LIN {X -85.223,Y -27.308,Z -231.114,A -90.000,B 90.000,C 0.000} C_DIS
LIN {X -83.227,Y -27.308,Z -229.864,A -90.000,B 90.000,C 0.000} C_DIS
LIN {X -79.994,Y -27.308,Z -227.837,A -90.000,B 90.000,C 0.000} C_DIS
LIN {X -76.849,Y -27.308,Z -225.880,A -90.000,B 90.000,C 0.000} C_DIS
LIN {X -68.403,Y -27.308,Z -220.902,A -90.000,B 90.000,C 0.000} C_DIS
LIN {X -66.455,Y -27.308,Z -219.796,A -90.000,B 90.000,C 0.000} C_DIS
LIN {X -60.717,Y -27.308,Z -216.545,A -90.000,B 90.000,C 0.000} C_DIS
LIN {X -59.585,Y -27.308,Z -215.913,A -90.000,B 90.000,C 0.000} C_DIS
LIN {X -54.120,Y -27.308,Z -212.892,A -90.000,B 90.000,C 0.000} C_DIS
LIN {X -51.972,Y -27.308,Z -211.724,A -90.000,B 90.000,C 0.000} C_DIS
LIN {X -46.281,Y -27.308,Z -208.611,A -90.000,B 90.000,C 0.000} C_DIS
LIN {X -44.940,Y -27.308,Z -207.894,A -90.000,B 90.000,C 0.000} C_DIS
LIN {X -41.211,Y -27.308,Z -205.831,A -90.000,B 90.000,C 0.000} C_DIS
LIN {X -39.138,Y -27.308,Z -204.699,A -90.000,B 90.000,C 0.000} C_DIS
LIN {X -36.802,Y -27.308,Z -203.366,A -90.000,B 90.000,C 0.000} C_DIS
LIN {X -34.331,Y -27.308,Z -201.960,A -90.000,B 90.000,C 0.000} C_DIS
LIN {X -30.365,Y -27.308,Z -199.567,A -90.000,B 90.000,C 0.000} C_DIS
LIN {X -27.103,Y -27.308,Z -197.441,A -90.000,B 90.000,C 0.000} C_DIS
LIN {X -24.362,Y -27.308,Z -195.502,A -90.000,B 90.000,C 0.000} C_DIS
LIN {X -23.811,Y -27.308,Z -195.108,A -90.000,B 90.000,C 0.000} C_DIS
LIN {X -22.633,Y -27.308,Z -194.200,A -90.000,B 90.000,C 0.000} C_DIS
LIN {X -20.957,Y -27.308,Z -192.878,A -90.000,B 90.000,C 0.000} C_DIS
LIN {X -19.924,Y -27.308,Z -192.013,A -90.000,B 90.000,C 0.000} C_DIS
LIN {X -17.934,Y -27.308,Z -190.290,A -90.000,B 90.000,C 0.000} C_DIS
LIN {X -17.733,Y -27.308,Z -190.109,A -90.000,B 90.000,C 0.000} C_DIS
LIN {X -15.439,Y -27.308,Z -187.960,A -90.000,B 90.000,C 0.000} C_DIS
LIN {X -15.234,Y -27.308,Z -187.762,A -90.000,B 90.000,C 0.000} C_DIS
LIN {X -13.962,Y -27.308,Z -186.449,A -90.000,B 90.000,C 0.000} C_DIS
LIN {X -12.177,Y -27.308,Z -184.664,A -90.000,B 90.000,C 0.000} C_DIS
LIN {X -10.066,Y -27.308,Z -182.306,A -90.000,B 90.000,C 0.000} C_DIS
LIN {X -9.477,Y -27.308,Z -181.655,A -90.000,B 90.000,C 0.000} C_DIS
LIN {X -7.788,Y -27.308,Z -179.586,A -90.000,B 90.000,C 0.000} C_DIS
LIN {X -6.794,Y -27.308,Z -178.283,A -90.000,B 90.000,C 0.000} C_DIS
LIN {X -6.582,Y -27.308,Z -177.987,A -90.000,B 90.000,C 0.000} C_DIS
LIN {X -6.159,Y -27.308,Z -177.338,A -90.000,B 90.000,C 0.000} C_DIS
LIN {X -4.783,Y -27.308,Z -175.273,A -90.000,B 90.000,C 0.000} C_DIS
LIN {X -4.713,Y -27.308,Z -175.159,A -90.000,B 90.000,C 0.000} C_DIS
LIN {X -3.540,Y -27.308,Z -173.039,A -90.000,B 90.000,C 0.000} C_DIS
LIN {X -2.865,Y -27.308,Z -171.671,A -90.000,B 90.000,C 0.000} C_DIS
LIN {X -2.832,Y -27.308,Z -171.590,A -90.000,B 90.000,C 0.000} C_DIS
LIN {X -2.604,Y -27.308,Z -170.921,A -90.000,B 90.000,C 0.000} C_DIS
LIN {X -1.680,Y -27.308,Z -168.354,A -90.000,B 90.000,C 0.000} C_DIS
LIN {X -1.356,Y -27.308,Z -166.665,A -90.000,B 90.000,C 0.000} C_DIS
LIN {X -1.145,Y -27.308,Z -165.329,A -90.000,B 90.000,C 0.000} C_DIS
LIN {X -1.146,Y -27.308,Z -165.323,A -90.000,B 90.000,C 0.000} C_DIS
LIN {X -1.174,Y -27.308,Z -164.878,A -90.000,B 90.000,C 0.000} C_DIS
LIN {X -1.320,Y -27.308,Z -162.962,A -90.000,B 90.000,C 0.000} C_DIS
LIN {X -1.678,Y -27.308,Z -162.121,A -90.000,B 90.000,C 0.000} C_DIS
LIN {X -2.018,Y -27.308,Z -161.227,A -90.000,B 90.000,C 0.000} C_DIS
LIN {X -2.779,Y -27.308,Z -160.228,A -90.000,B 90.000,C 0.000} C_DIS
LIN {X -3.012,Y -27.308,Z -159.916,A -90.000,B 90.000,C 0.000} C_DIS
LIN {X -3.062,Y -27.308,Z -159.845,A -90.000,B 90.000,C 0.000} C_DIS
LIN {X -3.809,Y -27.308,Z -159.198,A -90.000,B 90.000,C 0.000} C_DIS
LIN {X -4.494,Y -27.308,Z -158.553,A -90.000,B 90.000,C 0.000} C_DIS
LIN {X -5.258,Y -27.308,Z -158.041,A -90.000,B 90.000,C 0.000} C_DIS
LIN {X -6.409,Y -27.308,Z -157.185,A -90.000,B 90.000,C 0.000} C_DIS
LIN {X -7.420,Y -27.308,Z -156.518,A -90.000,B 90.000,C 0.000} C_DIS
LIN {X -8.434,Y -27.308,Z -155.815,A -90.000,B 90.000,C 0.000} C_DIS
LIN {X -8.921,Y -27.308,Z -155.486,A -90.000,B 90.000,C 0.000} C_DIS
LIN {X -10.919,Y -27.308,Z -154.124,A -90.000,B 90.000,C 0.000} C_DIS
LIN {X -11.534,Y -27.308,Z -153.660,A -90.000,B 90.000,C 0.000} C_DIS
LIN {X -13.381,Y -27.308,Z -152.360,A -90.000,B 90.000,C 0.000} C_DIS
LIN {X -13.865,Y -27.308,Z -151.978,A -90.000,B 90.000,C 0.000} C_DIS
LIN {X -16.164,Y -27.308,Z -150.260,A -90.000,B 90.000,C 0.000} C_DIS
LIN {X -16.733,Y -27.308,Z -149.790,A -90.000,B 90.000,C 0.000} C_DIS
LIN {X -18.323,Y -27.308,Z -148.512,A -90.000,B 90.000,C 0.000} C_DIS
LIN {X -18.612,Y -27.308,Z -148.282,A -90.000,B 90.000,C 0.000} C_DIS
LIN {X -19.226,Y -27.308,Z -147.818,A -90.000,B 90.000,C 0.000} C_DIS
LIN {X -19.599,Y -27.308,Z -147.522,A -90.000,B 90.000,C 0.000} C_DIS
LIN {X -20.909,Y -27.308,Z -146.394,A -90.000,B 90.000,C 0.000} C_DIS
LIN {X -22.705,Y -27.308,Z -144.892,A -90.000,B 90.000,C 0.000} C_DIS
LIN {X -23.016,Y -27.308,Z -144.647,A -90.000,B 90.000,C 0.000} C_DIS
LIN {X -24.434,Y -27.308,Z -143.351,A -90.000,B 90.000,C 0.000} C_DIS
LIN {X -25.785,Y -27.308,Z -142.145,A -90.000,B 90.000,C 0.000} C_DIS
LIN {X -26.430,Y -27.308,Z -141.592,A -90.000,B 90.000,C 0.000} C_DIS
LIN {X -26.511,Y -27.308,Z -141.523,A -90.000,B 90.000,C 0.000} C_DIS
LIN {X -26.798,Y -27.308,Z -141.263,A -90.000,B 90.000,C 0.000} C_DIS
LIN {X -27.182,Y -27.308,Z -140.891,A -90.000,B 90.000,C 0.000} C_DIS
LIN {X -30.222,Y -27.308,Z -137.840,A -90.000,B 90.000,C 0.000} C_DIS
LIN {X -30.546,Y -27.308,Z -137.455,A -90.000,B 90.000,C 0.000} C_DIS
LIN {X -32.740,Y -27.308,Z -134.749,A -90.000,B 90.000,C 0.000} C_DIS
LIN {X -33.314,Y -27.308,Z -134.051,A -90.000,B 90.000,C 0.000} C_DIS
LIN {X -33.612,Y -27.308,Z -133.614,A -90.000,B 90.000,C 0.000} C_DIS
LIN {X -35.907,Y -27.308,Z -130.179,A -90.000,B 90.000,C 0.000} C_DIS
LIN {X -37.258,Y -27.308,Z -127.712,A -90.000,B 90.000,C 0.000} C_DIS
LIN {X -37.397,Y -27.308,Z -127.454,A -90.000,B 90.000,C 0.000} C_DIS
LIN {X -38.165,Y -27.308,Z -126.016,A -90.000,B 90.000,C 0.000} C_DIS
LIN {X -38.975,Y -27.308,Z -124.190,A -90.000,B 90.000,C 0.000} C_DIS
LIN {X -39.648,Y -27.308,Z -122.652,A -90.000,B 90.000,C 0.000} C_DIS
LIN {X -39.793,Y -27.308,Z -122.312,A -90.000,B 90.000,C 0.000} C_DIS
LIN {X -40.196,Y -27.308,Z -121.317,A -90.000,B 90.000,C 0.000} C_DIS
LIN {X -40.311,Y -27.308,Z -120.980,A -90.000,B 90.000,C 0.000} C_DIS
LIN {X -40.482,Y -27.308,Z -120.456,A -90.000,B 90.000,C 0.000} C_DIS
LIN {X -40.902,Y -27.308,Z -119.024,A -90.000,B 90.000,C 0.000} C_DIS
LIN {X -41.166,Y -27.308,Z -118.090,A -90.000,B 90.000,C 0.000} C_DIS
LIN {X -41.278,Y -27.308,Z -117.687,A -90.000,B 90.000,C 0.000} C_DIS
LIN {X -41.299,Y -27.308,Z -117.605,A -90.000,B 90.000,C 0.000} C_DIS
LIN {X -41.911,Y -27.308,Z -115.570,A -90.000,B 90.000,C 0.000} C_DIS
LIN {X -42.357,Y -27.308,Z -114.398,A -90.000,B 90.000,C 0.000} C_DIS
LIN {X -42.549,Y -27.308,Z -113.916,A -90.000,B 90.000,C 0.000} C_DIS
LIN {X -43.092,Y -27.308,Z -112.840,A -90.000,B 90.000,C 0.000} C_DIS
LIN {X -43.558,Y -27.308,Z -111.969,A -90.000,B 90.000,C 0.000} C_DIS
LIN {X -44.072,Y -27.308,Z -111.153,A -90.000,B 90.000,C 0.000} C_DIS
LIN {X -45.121,Y -27.308,Z -109.594,A -90.000,B 90.000,C 0.000} C_DIS
LIN {X -45.338,Y -27.308,Z -109.287,A -90.000,B 90.000,C 0.000} C_DIS
LIN {X -46.992,Y -27.308,Z -107.075,A -90.000,B 90.000,C 0.000} C_DIS
LIN {X -47.098,Y -27.308,Z -106.927,A -90.000,B 90.000,C 0.000} C_DIS
LIN {X -48.585,Y -27.308,Z -104.967,A -90.000,B 90.000,C 0.000} C_DIS
LIN {X -49.203,Y -27.308,Z -104.208,A -90.000,B 90.000,C 0.000} C_DIS
LIN {X -49.940,Y -27.308,Z -103.250,A -90.000,B 90.000,C 0.000} C_DIS
LIN {X -51.313,Y -27.308,Z -101.558,A -90.000,B 90.000,C 0.000} C_DIS
LIN {X -51.724,Y -27.308,Z -101.045,A -90.000,B 90.000,C 0.000} C_DIS
LIN {X -53.185,Y -27.308,Z -99.120,A -90.000,B 90.000,C 0.000} C_DIS
LIN {X -53.957,Y -27.308,Z -98.076,A -90.000,B 90.000,C 0.000} C_DIS
LIN {X -54.226,Y -27.308,Z -97.727,A -90.000,B 90.000,C 0.000} C_DIS
LIN {X -55.529,Y -27.308,Z -95.927,A -90.000,B 90.000,C 0.000} C_DIS
LIN {X -56.485,Y -27.308,Z -94.658,A -90.000,B 90.000,C 0.000} C_DIS
LIN {X -56.867,Y -27.308,Z -94.134,A -90.000,B 90.000,C 0.000} C_DIS
LIN {X -58.660,Y -27.308,Z -91.749,A -90.000,B 90.000,C 0.000} C_DIS
LIN {X -58.816,Y -27.308,Z -91.546,A -90.000,B 90.000,C 0.000} C_DIS
LIN {X -60.216,Y -27.308,Z -89.639,A -90.000,B 90.000,C 0.000} C_DIS
LIN {X -60.437,Y -27.308,Z -89.333,A -90.000,B 90.000,C 0.000} C_DIS
LIN {X -60.531,Y -27.308,Z -89.209,A -90.000,B 90.000,C 0.000} C_DIS
LIN {X -61.646,Y -27.308,Z -87.834,A -90.000,B 90.000,C 0.000} C_DIS
LIN {X -62.365,Y -27.308,Z -86.929,A -90.000,B 90.000,C 0.000} C_DIS
LIN {X -63.967,Y -27.308,Z -85.103,A -90.000,B 90.000,C 0.000} C_DIS
LIN {X -64.183,Y -27.308,Z -84.856,A -90.000,B 90.000,C 0.000} C_DIS
LIN {X -65.298,Y -27.308,Z -83.619,A -90.000,B 90.000,C 0.000} C_DIS
LIN {X -65.834,Y -27.308,Z -82.993,A -90.000,B 90.000,C 0.000} C_DIS
LIN {X -66.748,Y -27.308,Z -81.917,A -90.000,B 90.000,C 0.000} C_DIS
LIN {X -67.132,Y -27.308,Z -81.454,A -90.000,B 90.000,C 0.000} C_DIS
LIN {X -67.558,Y -27.308,Z -80.989,A -90.000,B 90.000,C 0.000} C_DIS
LIN {X -68.611,Y -27.308,Z -79.786,A -90.000,B 90.000,C 0.000} C_DIS
LIN {X -69.303,Y -27.308,Z -78.987,A -90.000,B 90.000,C 0.000} C_DIS
LIN {X -69.822,Y -27.308,Z -78.380,A -90.000,B 90.000,C 0.000} C_DIS
LIN {X -70.935,Y -27.308,Z -77.008,A -90.000,B 90.000,C 0.000} C_DIS
LIN {X -71.960,Y -27.308,Z -75.857,A -90.000,B 90.000,C 0.000} C_DIS
LIN {X -72.414,Y -27.308,Z -75.329,A -90.000,B 90.000,C 0.000} C_DIS
LIN {X -73.458,Y -27.308,Z -74.204,A -90.000,B 90.000,C 0.000} C_DIS
LIN {X -73.957,Y -27.308,Z -73.750,A -90.000,B 90.000,C 0.000} C_DIS
LIN {X -74.254,Y -27.308,Z -73.492,A -90.000,B 90.000,C 0.000} C_DIS
LIN {X -74.565,Y -27.308,Z -73.279,A -90.000,B 90.000,C 0.000} C_DIS
LIN {X -74.767,Y -27.308,Z -73.138,A -90.000,B 90.000,C 0.000} C_DIS
LIN {X -74.798,Y -27.308,Z -73.125,A -90.000,B 90.000,C 0.000} C_DIS
LIN {X -75.017,Y -27.308,Z -73.097,A -90.000,B 90.000,C 0.000} C_DIS
LIN {X -75.670,Y -27.308,Z -73.073,A -90.000,B 90.000,C 0.000} C_DIS
LIN {X -76.020,Y -27.308,Z -73.070,A -90.000,B 90.000,C 0.000} C_DIS
LIN {X -76.334,Y -27.308,Z -73.065,A -90.000,B 90.000,C 0.000} C_DIS
LIN {X -76.599,Y -27.308,Z -73.057,A -90.000,B 90.000,C 0.000} C_DIS
LIN {X -76.851,Y -27.308,Z -73.043,A -90.000,B 90.000,C 0.000} C_DIS
LIN {X -77.230,Y -27.308,Z -73.013,A -90.000,B 90.000,C 0.000} C_DIS
LIN {X -77.574,Y -27.308,Z -72.983,A -90.000,B 90.000,C 0.000} C_DIS
LIN {X -77.718,Y -27.308,Z -72.968,A -90.000,B 90.000,C 0.000} C_DIS
LIN {X -78.228,Y -27.308,Z -72.885,A -90.000,B 90.000,C 0.000} C_DIS
LIN {X -78.608,Y -27.308,Z -72.796,A -90.000,B 90.000,C 0.000} C_DIS
LIN {X -78.915,Y -27.308,Z -72.710,A -90.000,B 90.000,C 0.000} C_DIS
LIN {X -79.319,Y -27.308,Z -72.586,A -90.000,B 90.000,C 0.000} C_DIS
LIN {X -79.675,Y -27.308,Z -72.471,A -90.000,B 90.000,C 0.000} C_DIS
LIN {X -80.019,Y -27.308,Z -72.348,A -90.000,B 90.000,C 0.000} C_DIS
LIN {X -80.375,Y -27.308,Z -72.185,A -90.000,B 90.000,C 0.000} C_DIS
LIN {X -80.697,Y -27.308,Z -72.027,A -90.000,B 90.000,C 0.000} C_DIS
LIN {X -80.992,Y -27.308,Z -71.848,A -90.000,B 90.000,C 0.000} C_DIS
LIN {X -81.324,Y -27.308,Z -71.641,A -90.000,B 90.000,C 0.000} C_DIS
LIN {X -81.637,Y -27.308,Z -71.388,A -90.000,B 90.000,C 0.000} C_DIS
LIN {X -81.835,Y -27.308,Z -71.211,A -90.000,B 90.000,C 0.000} C_DIS
LIN {X -82.059,Y -27.308,Z -71.022,A -90.000,B 90.000,C 0.000} C_DIS
LIN {X -82.156,Y -27.308,Z -70.939,A -90.000,B 90.000,C 0.000} C_DIS
LIN {X -82.435,Y -27.308,Z -70.649,A -90.000,B 90.000,C 0.000} C_DIS
LIN {X -82.682,Y -27.308,Z -70.318,A -90.000,B 90.000,C 0.000} C_DIS
LIN {X -82.800,Y -27.308,Z -70.155,A -90.000,B 90.000,C 0.000} C_DIS
LIN {X -82.856,Y -27.308,Z -70.085,A -90.000,B 90.000,C 0.000} C_DIS
LIN {X -83.029,Y -27.308,Z -69.840,A -90.000,B 90.000,C 0.000} C_DIS
LIN {X -83.229,Y -27.308,Z -69.490,A -90.000,B 90.000,C 0.000} C_DIS
LIN {X -83.356,Y -27.308,Z -69.184,A -90.000,B 90.000,C 0.000} C_DIS
LIN {X -83.500,Y -27.308,Z -68.887,A -90.000,B 90.000,C 0.000} C_DIS
LIN {X -83.522,Y -27.308,Z -68.835,A -90.000,B 90.000,C 0.000} C_DIS
LIN {X -83.644,Y -27.308,Z -68.492,A -90.000,B 90.000,C 0.000} C_DIS
LIN {X -83.662,Y -27.308,Z -68.425,A -90.000,B 90.000,C 0.000} C_DIS
LIN {X -83.731,Y -27.308,Z -68.129,A -90.000,B 90.000,C 0.000} C_DIS
LIN {X -83.778,Y -27.308,Z -67.975,A -90.000,B 90.000,C 0.000} C_DIS
LIN {X -83.872,Y -27.308,Z -67.562,A -90.000,B 90.000,C 0.000} C_DIS
LIN {X -83.897,Y -27.308,Z -67.322,A -90.000,B 90.000,C 0.000} C_DIS
LIN {X -84.004,Y -27.308,Z -66.971,A -90.000,B 90.000,C 0.000} C_DIS
LIN {X -84.037,Y -27.308,Z -66.849,A -90.000,B 90.000,C 0.000} C_DIS
LIN {X -84.152,Y -27.308,Z -66.309,A -90.000,B 90.000,C 0.000} C_DIS
LIN {X -84.180,Y -27.308,Z -66.154,A -90.000,B 90.000,C 0.000} C_DIS
LIN {X -84.260,Y -27.308,Z -65.657,A -90.000,B 90.000,C 0.000} C_DIS
LIN {X -84.279,Y -27.308,Z -65.543,A -90.000,B 90.000,C 0.000} C_DIS
LIN {X -84.322,Y -27.308,Z -65.297,A -90.000,B 90.000,C 0.000} C_DIS
LIN {X -84.357,Y -27.308,Z -65.124,A -90.000,B 90.000,C 0.000} C_DIS
LIN {X -84.404,Y -27.308,Z -64.967,A -90.000,B 90.000,C 0.000} C_DIS
LIN {X -84.600,Y -27.308,Z -64.383,A -90.000,B 90.000,C 0.000} C_DIS
LIN {X -84.702,Y -27.308,Z -64.055,A -90.000,B 90.000,C 0.000} C_DIS
LIN {X -84.904,Y -27.308,Z -63.276,A -90.000,B 90.000,C 0.000} C_DIS
LIN {X -84.929,Y -27.308,Z -63.196,A -90.000,B 90.000,C 0.000} C_DIS
LIN {X -84.968,Y -27.308,Z -63.107,A -90.000,B 90.000,C 0.000} C_DIS
LIN {X -85.046,Y -27.308,Z -62.905,A -90.000,B 90.000,C 0.000} C_DIS
LIN {X -85.068,Y -27.308,Z -62.858,A -90.000,B 90.000,C 0.000} C_DIS
LIN {X -85.176,Y -27.308,Z -62.700,A -90.000,B 90.000,C 0.000} C_DIS
LIN {X -85.293,Y -27.308,Z -62.562,A -90.000,B 90.000,C 0.000} C_DIS
LIN {X -85.630,Y -27.308,Z -62.148,A -90.000,B 90.000,C 0.000} C_DIS
LIN {X -86.250,Y -27.308,Z -61.521,A -90.000,B 90.000,C 0.000} C_DIS
LIN {X -86.385,Y -27.308,Z -61.384,A -90.000,B 90.000,C 0.000} C_DIS
LIN {X -86.893,Y -27.308,Z -60.912,A -90.000,B 90.000,C 0.000} C_DIS
LIN {X -87.654,Y -27.308,Z -60.199,A -90.000,B 90.000,C 0.000} C_DIS
LIN {X -88.400,Y -27.308,Z -59.530,A -90.000,B 90.000,C 0.000} C_DIS
LIN {X -89.022,Y -27.308,Z -58.966,A -90.000,B 90.000,C 0.000} C_DIS
LIN {X -89.404,Y -27.308,Z -58.604,A -90.000,B 90.000,C 0.000} C_DIS
LIN {X -90.679,Y -27.308,Z -57.368,A -90.000,B 90.000,C 0.000} C_DIS
LIN {X -90.874,Y -27.308,Z -57.173,A -90.000,B 90.000,C 0.000} C_DIS
LIN {X -91.295,Y -27.308,Z -56.741,A -90.000,B 90.000,C 0.000} C_DIS
LIN {X -91.759,Y -27.308,Z -56.238,A -90.000,B 90.000,C 0.000} C_DIS
LIN {X -92.620,Y -27.308,Z -55.242,A -90.000,B 90.000,C 0.000} C_DIS
LIN {X -93.104,Y -27.308,Z -54.609,A -90.000,B 90.000,C 0.000} C_DIS
LIN {X -93.380,Y -27.308,Z -54.235,A -90.000,B 90.000,C 0.000} C_DIS
LIN {X -93.514,Y -27.308,Z -54.050,A -90.000,B 90.000,C 0.000} C_DIS
LIN {X -93.898,Y -27.308,Z -53.393,A -90.000,B 90.000,C 0.000} C_DIS
LIN {X -93.958,Y -27.308,Z -53.276,A -90.000,B 90.000,C 0.000} C_DIS
LIN {X -94.142,Y -27.308,Z -52.904,A -90.000,B 90.000,C 0.000} C_DIS
LIN {X -94.334,Y -27.308,Z -52.418,A -90.000,B 90.000,C 0.000} C_DIS
LIN {X -94.397,Y -27.308,Z -52.255,A -90.000,B 90.000,C 0.000} C_DIS
LIN {X -94.572,Y -27.308,Z -51.708,A -90.000,B 90.000,C 0.000} C_DIS
LIN {X -94.624,Y -27.308,Z -51.540,A -90.000,B 90.000,C 0.000} C_DIS
LIN {X -94.663,Y -27.308,Z -51.261,A -90.000,B 90.000,C 0.000} C_DIS
LIN {X -94.690,Y -27.308,Z -50.989,A -90.000,B 90.000,C 0.000} C_DIS
LIN {X -94.708,Y -27.308,Z -50.849,A -90.000,B 90.000,C 0.000} C_DIS
LIN {X -94.705,Y -27.308,Z -50.520,A -90.000,B 90.000,C 0.000} C_DIS
LIN {X -94.685,Y -27.308,Z -50.284,A -90.000,B 90.000,C 0.000} C_DIS
LIN {X -94.633,Y -27.308,Z -49.971,A -90.000,B 90.000,C 0.000} C_DIS
LIN {X -94.628,Y -27.308,Z -49.914,A -90.000,B 90.000,C 0.000} C_DIS
LIN {X -94.559,Y -27.308,Z -49.687,A -90.000,B 90.000,C 0.000} C_DIS
LIN {X -94.426,Y -27.308,Z -49.421,A -90.000,B 90.000,C 0.000} C_DIS
LIN {X -94.404,Y -27.308,Z -49.356,A -90.000,B 90.000,C 0.000} C_DIS
LIN {X -94.289,Y -27.308,Z -49.148,A -90.000,B 90.000,C 0.000} C_DIS
LIN {X -94.134,Y -27.308,Z -48.970,A -90.000,B 90.000,C 0.000} C_DIS
LIN {X -94.079,Y -27.308,Z -48.910,A -90.000,B 90.000,C 0.000} C_DIS
LIN {X -94.043,Y -27.308,Z -48.853,A -90.000,B 90.000,C 0.000} C_DIS
LIN {X -93.887,Y -27.308,Z -48.674,A -90.000,B 90.000,C 0.000} C_DIS
LIN {X -93.617,Y -27.308,Z -48.473,A -90.000,B 90.000,C 0.000} C_DIS
LIN {X -93.557,Y -27.308,Z -48.413,A -90.000,B 90.000,C 0.000} C_DIS
LIN {X -93.414,Y -27.308,Z -48.295,A -90.000,B 90.000,C 0.000} C_DIS
LIN {X -93.204,Y -27.308,Z -48.138,A -90.000,B 90.000,C 0.000} C_DIS
LIN {X -92.952,Y -27.308,Z -48.011,A -90.000,B 90.000,C 0.000} C_DIS
LIN {X -92.775,Y -27.308,Z -47.952,A -90.000,B 90.000,C 0.000} C_DIS
LIN {X -92.483,Y -27.308,Z -47.821,A -90.000,B 90.000,C 0.000} C_DIS
LIN {X -92.213,Y -27.308,Z -47.741,A -90.000,B 90.000,C 0.000} C_DIS
LIN {X -91.652,Y -27.308,Z -47.616,A -90.000,B 90.000,C 0.000} C_DIS
LIN {X -91.311,Y -27.308,Z -47.593,A -90.000,B 90.000,C 0.000} C_DIS
LIN {X -90.543,Y -27.308,Z -47.616,A -90.000,B 90.000,C 0.000} C_DIS
LIN {X -90.225,Y -27.308,Z -47.643,A -90.000,B 90.000,C 0.000} C_DIS
LIN {X -89.409,Y -27.308,Z -47.720,A -90.000,B 90.000,C 0.000} C_DIS
LIN {X -88.277,Y -27.308,Z -47.951,A -90.000,B 90.000,C 0.000} C_DIS
LIN {X -88.112,Y -27.308,Z -47.999,A -90.000,B 90.000,C 0.000} C_DIS
LIN {X -86.815,Y -27.308,Z -48.411,A -90.000,B 90.000,C 0.000} C_DIS
LIN {X -86.455,Y -27.308,Z -48.530,A -90.000,B 90.000,C 0.000} C_DIS
LIN {X -85.645,Y -27.308,Z -48.823,A -90.000,B 90.000,C 0.000} C_DIS
LIN {X -85.388,Y -27.308,Z -48.929,A -90.000,B 90.000,C 0.000} C_DIS
LIN {X -84.854,Y -27.308,Z -49.164,A -90.000,B 90.000,C 0.000} C_DIS
LIN {X -82.923,Y -27.308,Z -50.118,A -90.000,B 90.000,C 0.000} C_DIS
LIN {X -82.842,Y -27.308,Z -50.159,A -90.000,B 90.000,C 0.000} C_DIS
LIN {X -81.799,Y -27.308,Z -50.772,A -90.000,B 90.000,C 0.000} C_DIS
LIN {X -80.820,Y -27.308,Z -51.324,A -90.000,B 90.000,C 0.000} C_DIS
LIN {X -80.098,Y -27.308,Z -51.785,A -90.000,B 90.000,C 0.000} C_DIS
LIN {X -79.415,Y -27.308,Z -52.233,A -90.000,B 90.000,C 0.000} C_DIS
LIN {X -78.943,Y -27.308,Z -52.512,A -90.000,B 90.000,C 0.000} C_DIS
LIN {X -78.820,Y -27.308,Z -52.591,A -90.000,B 90.000,C 0.000} C_DIS
LIN {X -78.713,Y -27.308,Z -52.652,A -90.000,B 90.000,C 0.000} C_DIS
LIN {X -78.353,Y -27.308,Z -52.874,A -90.000,B 90.000,C 0.000} C_DIS
LIN {X -78.152,Y -27.308,Z -52.915,A -90.000,B 90.000,C 0.000} C_DIS
LIN {X -77.685,Y -27.308,Z -52.891,A -90.000,B 90.000,C 0.000} C_DIS
LIN {X -77.521,Y -27.308,Z -52.843,A -90.000,B 90.000,C 0.000} C_DIS
LIN {X -76.977,Y -27.308,Z -52.661,A -90.000,B 90.000,C 0.000} C_DIS
LIN {X -76.822,Y -27.308,Z -52.584,A -90.000,B 90.000,C 0.000} C_DIS
LIN {X -76.230,Y -27.308,Z -52.231,A -90.000,B 90.000,C 0.000} C_DIS
LIN {X -75.911,Y -27.308,Z -51.880,A -90.000,B 90.000,C 0.000} C_DIS
LIN {X -75.721,Y -27.308,Z -51.738,A -90.000,B 90.000,C 0.000} C_DIS
LIN {X -75.688,Y -27.308,Z -51.716,A -90.000,B 90.000,C 0.000} C_DIS
LIN {X -75.432,Y -27.308,Z -51.196,A -90.000,B 90.000,C 0.000} C_DIS
LIN {X -75.358,Y -27.308,Z -51.059,A -90.000,B 90.000,C 0.000} C_DIS
LIN {X -75.315,Y -27.308,Z -51.015,A -90.000,B 90.000,C 0.000} C_DIS
LIN {X -75.268,Y -27.308,Z -50.824,A -90.000,B 90.000,C 0.000} C_DIS
LIN {X -75.257,Y -27.308,Z -50.431,A -90.000,B 90.000,C 0.000} C_DIS
LIN {X -75.437,Y -27.308,Z -49.585,A -90.000,B 90.000,C 0.000} C_DIS
LIN {X -75.451,Y -27.308,Z -49.419,A -90.000,B 90.000,C 0.000} C_DIS
LIN {X -75.470,Y -27.308,Z -49.322,A -90.000,B 90.000,C 0.000} C_DIS
LIN {X -75.528,Y -27.308,Z -48.845,A -90.000,B 90.000,C 0.000} C_DIS
LIN {X -75.614,Y -27.308,Z -48.700,A -90.000,B 90.000,C 0.000} C_DIS
LIN {X -75.778,Y -27.308,Z -48.315,A -90.000,B 90.000,C 0.000} C_DIS
LIN {X -75.772,Y -27.308,Z -48.226,A -90.000,B 90.000,C 0.000} C_DIS
LIN {X -75.702,Y -27.308,Z -48.112,A -90.000,B 90.000,C 0.000} C_DIS
LIN {X -75.670,Y -27.308,Z -47.358,A -90.000,B 90.000,C 0.000} C_DIS
LIN {X -75.666,Y -27.308,Z -47.285,A -90.000,B 90.000,C 0.000} C_DIS
LIN {X -75.614,Y -27.308,Z -47.213,A -90.000,B 90.000,C 0.000} C_DIS
LIN {X -75.532,Y -27.308,Z -47.179,A -90.000,B 90.000,C 0.000} C_DIS
LIN {X -74.785,Y -27.308,Z -46.921,A -90.000,B 90.000,C 0.000} C_DIS
LIN {X -74.518,Y -27.308,Z -46.858,A -90.000,B 90.000,C 0.000} C_DIS
LIN {X -74.497,Y -27.308,Z -46.853,A -90.000,B 90.000,C 0.000} C_DIS
LIN {X -74.317,Y -27.308,Z -46.860,A -90.000,B 90.000,C 0.000} C_DIS
LIN {X -74.256,Y -27.308,Z -46.876,A -90.000,B 90.000,C 0.000} C_DIS
LIN {X -72.929,Y -27.308,Z -47.028,A -90.000,B 90.000,C 0.000} C_DIS
LIN {X -72.759,Y -27.308,Z -47.084,A -90.000,B 90.000,C 0.000} C_DIS
LIN {X -72.617,Y -27.308,Z -47.137,A -90.000,B 90.000,C 0.000} C_DIS
LIN {X -71.380,Y -27.308,Z -47.421,A -90.000,B 90.000,C 0.000} C_DIS
LIN {X -71.211,Y -27.308,Z -47.477,A -90.000,B 90.000,C 0.000} C_DIS
LIN {X -71.067,Y -27.308,Z -47.534,A -90.000,B 90.000,C 0.000} C_DIS
LIN {X -69.599,Y -27.308,Z -47.870,A -90.000,B 90.000,C 0.000} C_DIS
LIN {X -69.349,Y -27.308,Z -47.873,A -90.000,B 90.000,C 0.000} C_DIS
LIN {X -67.886,Y -27.308,Z -48.166,A -90.000,B 90.000,C 0.000} C_DIS
LIN {X -67.535,Y -27.308,Z -48.228,A -90.000,B 90.000,C 0.000} C_DIS
LIN {X -67.302,Y -27.308,Z -48.275,A -90.000,B 90.000,C 0.000} C_DIS
LIN {X -67.283,Y -27.308,Z -48.281,A -90.000,B 90.000,C 0.000} C_DIS
LIN {X -66.642,Y -27.308,Z -48.353,A -90.000,B 90.000,C 0.000} C_DIS
LIN {X -64.888,Y -27.308,Z -48.721,A -90.000,B 90.000,C 0.000} C_DIS
LIN {X -64.684,Y -27.308,Z -48.736,A -90.000,B 90.000,C 0.000} C_DIS
LIN {X -64.583,Y -27.308,Z -48.752,A -90.000,B 90.000,C 0.000} C_DIS
LIN {X -63.765,Y -27.308,Z -48.882,A -90.000,B 90.000,C 0.000} C_DIS
LIN {X -62.172,Y -27.308,Z -49.234,A -90.000,B 90.000,C 0.000} C_DIS
LIN {X -61.720,Y -27.308,Z -49.293,A -90.000,B 90.000,C 0.000} C_DIS
LIN {X -60.768,Y -27.308,Z -49.482,A -90.000,B 90.000,C 0.000} C_DIS
LIN {X -60.425,Y -27.308,Z -49.558,A -90.000,B 90.000,C 0.000} C_DIS
LIN {X -59.345,Y -27.308,Z -49.806,A -90.000,B 90.000,C 0.000} C_DIS
LIN {X -58.678,Y -27.308,Z -49.920,A -90.000,B 90.000,C 0.000} C_DIS
LIN {X -58.325,Y -27.308,Z -49.999,A -90.000,B 90.000,C 0.000} C_DIS
LIN {X -56.851,Y -27.308,Z -50.342,A -90.000,B 90.000,C 0.000} C_DIS
LIN {X -56.345,Y -27.308,Z -50.459,A -90.000,B 90.000,C 0.000} C_DIS
LIN {X -55.296,Y -27.308,Z -50.666,A -90.000,B 90.000,C 0.000} C_DIS
LIN {X -53.371,Y -27.308,Z -51.124,A -90.000,B 90.000,C 0.000} C_DIS
LIN {X -53.286,Y -27.308,Z -51.142,A -90.000,B 90.000,C 0.000} C_DIS
LIN {X -53.131,Y -27.308,Z -51.179,A -90.000,B 90.000,C 0.000} C_DIS
LIN {X -51.402,Y -27.308,Z -51.571,A -90.000,B 90.000,C 0.000} C_DIS
LIN {X -50.457,Y -27.308,Z -51.814,A -90.000,B 90.000,C 0.000} C_DIS
LIN {X -49.578,Y -27.308,Z -52.017,A -90.000,B 90.000,C 0.000} C_DIS
LIN {X -48.351,Y -27.308,Z -52.327,A -90.000,B 90.000,C 0.000} C_DIS
LIN {X -47.858,Y -27.308,Z -52.433,A -90.000,B 90.000,C 0.000} C_DIS
LIN {X -47.456,Y -27.308,Z -52.528,A -90.000,B 90.000,C 0.000} C_DIS
LIN {X -47.282,Y -27.308,Z -52.565,A -90.000,B 90.000,C 0.000} C_DIS
LIN {X -46.851,Y -27.308,Z -52.617,A -90.000,B 90.000,C 0.000} C_DIS
LIN {X -46.055,Y -27.308,Z -52.645,A -90.000,B 90.000,C 0.000} C_DIS
LIN {X -45.267,Y -27.308,Z -52.678,A -90.000,B 90.000,C 0.000} C_DIS
LIN {X -43.988,Y -27.308,Z -52.715,A -90.000,B 90.000,C 0.000} C_DIS
LIN {X -42.867,Y -27.308,Z -52.774,A -90.000,B 90.000,C 0.000} C_DIS
LIN {X -42.549,Y -27.308,Z -52.801,A -90.000,B 90.000,C 0.000} C_DIS
LIN {X -41.808,Y -27.308,Z -52.875,A -90.000,B 90.000,C 0.000} C_DIS
LIN {X -39.572,Y -27.308,Z -53.109,A -90.000,B 90.000,C 0.000} C_DIS
LIN {X -38.701,Y -27.308,Z -53.242,A -90.000,B 90.000,C 0.000} C_DIS
LIN {X -38.096,Y -27.308,Z -53.337,A -90.000,B 90.000,C 0.000} C_DIS
LIN {X -36.582,Y -27.308,Z -53.593,A -90.000,B 90.000,C 0.000} C_DIS
LIN {X -35.657,Y -27.308,Z -53.760,A -90.000,B 90.000,C 0.000} C_DIS
LIN {X -33.190,Y -27.308,Z -54.250,A -90.000,B 90.000,C 0.000} C_DIS
LIN {X -32.731,Y -27.308,Z -54.338,A -90.000,B 90.000,C 0.000} C_DIS
LIN {X -31.973,Y -27.308,Z -54.494,A -90.000,B 90.000,C 0.000} C_DIS
LIN {X -29.563,Y -27.308,Z -55.034,A -90.000,B 90.000,C 0.000} C_DIS
LIN {X -28.572,Y -27.308,Z -55.243,A -90.000,B 90.000,C 0.000} C_DIS
LIN {X -26.759,Y -27.308,Z -55.630,A -90.000,B 90.000,C 0.000} C_DIS
LIN {X -25.274,Y -27.308,Z -55.904,A -90.000,B 90.000,C 0.000} C_DIS
LIN {X -24.524,Y -27.308,Z -56.024,A -90.000,B 90.000,C 0.000} C_DIS
LIN {X -23.511,Y -27.308,Z -56.150,A -90.000,B 90.000,C 0.000} C_DIS
LIN {X -22.723,Y -27.308,Z -56.207,A -90.000,B 90.000,C 0.000} C_DIS
LIN {X -22.397,Y -27.308,Z -56.214,A -90.000,B 90.000,C 0.000} C_DIS
LIN {X -21.650,Y -27.308,Z -56.177,A -90.000,B 90.000,C 0.000} C_DIS
LIN {X -21.553,Y -27.308,Z -56.165,A -90.000,B 90.000,C 0.000} C_DIS
LIN {X -20.887,Y -27.308,Z -56.039,A -90.000,B 90.000,C 0.000} C_DIS
LIN {X -20.751,Y -27.308,Z -56.012,A -90.000,B 90.000,C 0.000} C_DIS
LIN {X -19.986,Y -27.308,Z -55.706,A -90.000,B 90.000,C 0.000} C_DIS
LIN {X -19.512,Y -27.308,Z -55.554,A -90.000,B 90.000,C 0.000} C_DIS
LIN {X -18.660,Y -27.308,Z -55.186,A -90.000,B 90.000,C 0.000} C_DIS
LIN {X -18.036,Y -27.308,Z -54.936,A -90.000,B 90.000,C 0.000} C_DIS
LIN {X -17.892,Y -27.308,Z -54.873,A -90.000,B 90.000,C 0.000} C_DIS
LIN {X -15.925,Y -27.308,Z -54.124,A -90.000,B 90.000,C 0.000} C_DIS
LIN {X -15.504,Y -27.308,Z -53.994,A -90.000,B 90.000,C 0.000} C_DIS
LIN {X -14.478,Y -27.308,Z -53.726,A -90.000,B 90.000,C 0.000} C_DIS
LIN {X -13.147,Y -27.308,Z -53.413,A -90.000,B 90.000,C 0.000} C_DIS
LIN {X -12.872,Y -27.308,Z -53.351,A -90.000,B 90.000,C 0.000} C_DIS
LIN {X -12.439,Y -27.308,Z -53.269,A -90.000,B 90.000,C 0.000} C_DIS
LIN {X -12.071,Y -27.308,Z -53.231,A -90.000,B 90.000,C 0.000} C_DIS
LIN {X -11.636,Y -27.308,Z -53.190,A -90.000,B 90.000,C 0.000} C_DIS
LIN {X -11.196,Y -27.308,Z -53.158,A -90.000,B 90.000,C 0.000} C_DIS
LIN {X -10.086,Y -27.308,Z -53.119,A -90.000,B 90.000,C 0.000} C_DIS
LIN {X -9.111,Y -27.308,Z -53.076,A -90.000,B 90.000,C 0.000} C_DIS
LIN {X -8.324,Y -27.308,Z -53.066,A -90.000,B 90.000,C 0.000} C_DIS
LIN {X -8.178,Y -27.308,Z -53.071,A -90.000,B 90.000,C 0.000} C_DIS
LIN {X -7.941,Y -27.308,Z -53.086,A -90.000,B 90.000,C 0.000} C_DIS
LIN {X -5.929,Y -27.308,Z -53.244,A -90.000,B 90.000,C 0.000} C_DIS
LIN {X -5.507,Y -27.308,Z -53.284,A -90.000,B 90.000,C 0.000} C_DIS
LIN {X -2.491,Y -27.308,Z -53.719,A -90.000,B 90.000,C 0.000} C_DIS
LIN {X -0.877,Y -27.308,Z -54.086,A -90.000,B 90.000,C 0.000} C_DIS
LIN {X -0.384,Y -27.308,Z -54.174,A -90.000,B 90.000,C 0.000} C_DIS
LIN {X 0.435,Y -27.308,Z -54.334,A -90.000,B 90.000,C 0.000} C_DIS
LIN {X 1.127,Y -27.308,Z -54.517,A -90.000,B 90.000,C 0.000} C_DIS
LIN {X 2.471,Y -27.308,Z -54.795,A -90.000,B 90.000,C 0.000} C_DIS
LIN {X 2.756,Y -27.308,Z -54.869,A -90.000,B 90.000,C 0.000} C_DIS
LIN {X 4.090,Y -27.308,Z -55.127,A -90.000,B 90.000,C 0.000} C_DIS
LIN {X 4.736,Y -27.308,Z -55.198,A -90.000,B 90.000,C 0.000} C_DIS
LIN {X 5.276,Y -27.308,Z -55.272,A -90.000,B 90.000,C 0.000} C_DIS
LIN {X 5.687,Y -27.308,Z -55.287,A -90.000,B 90.000,C 0.000} C_DIS
LIN {X 6.858,Y -27.308,Z -55.282,A -90.000,B 90.000,C 0.000} C_DIS
LIN {X 7.864,Y -27.308,Z -55.201,A -90.000,B 90.000,C 0.000} C_DIS
LIN {X 8.134,Y -27.308,Z -55.173,A -90.000,B 90.000,C 0.000} C_DIS
LIN {X 9.252,Y -27.308,Z -55.047,A -90.000,B 90.000,C 0.000} C_DIS
LIN {X 9.652,Y -27.308,Z -55.015,A -90.000,B 90.000,C 0.000} C_DIS
LIN {X 9.923,Y -27.308,Z -54.998,A -90.000,B 90.000,C 0.000} C_DIS
LIN {X 11.157,Y -27.308,Z -55.007,A -90.000,B 90.000,C 0.000} C_DIS
LIN {X 11.508,Y -27.308,Z -55.034,A -90.000,B 90.000,C 0.000} C_DIS
LIN {X 12.331,Y -27.308,Z -55.162,A -90.000,B 90.000,C 0.000} C_DIS
LIN {X 12.569,Y -27.308,Z -55.172,A -90.000,B 90.000,C 0.000} C_DIS
LIN {X 12.876,Y -27.308,Z -55.188,A -90.000,B 90.000,C 0.000} C_DIS
LIN {X 13.561,Y -27.308,Z -55.299,A -90.000,B 90.000,C 0.000} C_DIS
LIN {X 14.134,Y -27.308,Z -55.349,A -90.000,B 90.000,C 0.000} C_DIS
LIN {X 14.781,Y -27.308,Z -55.438,A -90.000,B 90.000,C 0.000} C_DIS
LIN {X 15.213,Y -27.308,Z -55.466,A -90.000,B 90.000,C 0.000} C_DIS
LIN {X 15.445,Y -27.308,Z -55.493,A -90.000,B 90.000,C 0.000} C_DIS
LIN {X 15.887,Y -27.308,Z -55.507,A -90.000,B 90.000,C 0.000} C_DIS
LIN {X 16.274,Y -27.308,Z -55.547,A -90.000,B 90.000,C 0.000} C_DIS
LIN {X 16.722,Y -27.308,Z -55.556,A -90.000,B 90.000,C 0.000} C_DIS
LIN {X 17.040,Y -27.308,Z -55.597,A -90.000,B 90.000,C 0.000} C_DIS
LIN {X 17.121,Y -27.308,Z -55.600,A -90.000,B 90.000,C 0.000} C_DIS
LIN {X 17.542,Y -27.308,Z -55.641,A -90.000,B 90.000,C 0.000} C_DIS
LIN {X 17.858,Y -27.308,Z -55.690,A -90.000,B 90.000,C 0.000} C_DIS
LIN {X 18.015,Y -27.308,Z -55.721,A -90.000,B 90.000,C 0.000} C_DIS
LIN {X 18.204,Y -27.308,Z -55.741,A -90.000,B 90.000,C 0.000} C_DIS
LIN {X 18.617,Y -27.308,Z -55.830,A -90.000,B 90.000,C 0.000} C_DIS
LIN {X 19.037,Y -27.308,Z -55.956,A -90.000,B 90.000,C 0.000} C_DIS
LIN {X 19.207,Y -27.308,Z -55.994,A -90.000,B 90.000,C 0.000} C_DIS
LIN {X 19.430,Y -27.308,Z -55.767,A -90.000,B 90.000,C 0.000} C_DIS
LIN {X 19.513,Y -27.308,Z -55.686,A -90.000,B 90.000,C 0.000} C_DIS
LIN {X 19.879,Y -27.308,Z -55.352,A -90.000,B 90.000,C 0.000} C_DIS
LIN {X 20.370,Y -27.308,Z -54.995,A -90.000,B 90.000,C 0.000} C_DIS
LIN {X 20.445,Y -27.308,Z -54.936,A -90.000,B 90.000,C 0.000} C_DIS
LIN {X 20.628,Y -27.308,Z -54.661,A -90.000,B 90.000,C 0.000} C_DIS
LIN {X 20.626,Y -27.308,Z -54.647,A -90.000,B 90.000,C 0.000} C_DIS
LIN {X 20.641,Y -27.308,Z -54.468,A -90.000,B 90.000,C 0.000} C_DIS
LIN {X 20.652,Y -27.308,Z -54.145,A -90.000,B 90.000,C 0.000} C_DIS
LIN {X 20.672,Y -27.308,Z -53.909,A -90.000,B 90.000,C 0.000} C_DIS
LIN {X 20.840,Y -27.308,Z -53.367,A -90.000,B 90.000,C 0.000} C_DIS
LIN {X 21.056,Y -27.308,Z -52.822,A -90.000,B 90.000,C 0.000} C_DIS
LIN {X 21.165,Y -27.308,Z -52.561,A -90.000,B 90.000,C 0.000} C_DIS
LIN {X 21.317,Y -27.308,Z -52.324,A -90.000,B 90.000,C 0.000} C_DIS
LIN {X 21.558,Y -27.308,Z -51.960,A -90.000,B 90.000,C 0.000} C_DIS
LIN {X 21.711,Y -27.308,Z -51.723,A -90.000,B 90.000,C 0.000} C_DIS
LIN {X 21.853,Y -27.308,Z -51.536,A -90.000,B 90.000,C 0.000} C_DIS
LIN {X 21.956,Y -27.308,Z -51.381,A -90.000,B 90.000,C 0.000} C_DIS
LIN {X 22.023,Y -27.308,Z -51.285,A -90.000,B 90.000,C 0.000} C_DIS
LIN {X 22.445,Y -27.308,Z -50.799,A -90.000,B 90.000,C 0.000} C_DIS
LIN {X 22.741,Y -27.308,Z -50.473,A -90.000,B 90.000,C 0.000} C_DIS
LIN {X 22.835,Y -27.308,Z -50.383,A -90.000,B 90.000,C 0.000} C_DIS
LIN {X 23.027,Y -27.308,Z -50.153,A -90.000,B 90.000,C 0.000} C_DIS
LIN {X 23.258,Y -27.308,Z -49.924,A -90.000,B 90.000,C 0.000} C_DIS
LIN {X 23.576,Y -27.308,Z -49.598,A -90.000,B 90.000,C 0.000} C_DIS
LIN {X 23.818,Y -27.308,Z -49.361,A -90.000,B 90.000,C 0.000} C_DIS
LIN {X 23.864,Y -27.308,Z -49.321,A -90.000,B 90.000,C 0.000} C_DIS
LIN {X 24.021,Y -27.308,Z -49.140,A -90.000,B 90.000,C 0.000} C_DIS
LIN {X 24.598,Y -27.308,Z -48.590,A -90.000,B 90.000,C 0.000} C_DIS
LIN {X 24.869,Y -27.308,Z -48.344,A -90.000,B 90.000,C 0.000} C_DIS
LIN {X 24.954,Y -27.308,Z -48.272,A -90.000,B 90.000,C 0.000} C_DIS
LIN {X 25.011,Y -27.308,Z -48.211,A -90.000,B 90.000,C 0.000} C_DIS
LIN {X 25.672,Y -27.308,Z -47.627,A -90.000,B 90.000,C 0.000} C_DIS
LIN {X 25.884,Y -27.308,Z -47.452,A -90.000,B 90.000,C 0.000} C_DIS
LIN {X 26.341,Y -27.308,Z -47.101,A -90.000,B 90.000,C 0.000} C_DIS
LIN {X 26.504,Y -27.308,Z -46.986,A -90.000,B 90.000,C 0.000} C_DIS
LIN {X 26.644,Y -27.308,Z -46.866,A -90.000,B 90.000,C 0.000} C_DIS
LIN {X 26.996,Y -27.308,Z -46.604,A -90.000,B 90.000,C 0.000} C_DIS
LIN {X 27.661,Y -27.308,Z -46.179,A -90.000,B 90.000,C 0.000} C_DIS
LIN {X 28.096,Y -27.308,Z -45.955,A -90.000,B 90.000,C 0.000} C_DIS
LIN {X 28.319,Y -27.308,Z -45.835,A -90.000,B 90.000,C 0.000} C_DIS
LIN {X 28.417,Y -27.308,Z -45.791,A -90.000,B 90.000,C 0.000} C_DIS
LIN {X 29.159,Y -27.308,Z -45.424,A -90.000,B 90.000,C 0.000} C_DIS
LIN {X 29.587,Y -27.308,Z -45.239,A -90.000,B 90.000,C 0.000} C_DIS
LIN {X 30.107,Y -27.308,Z -45.056,A -90.000,B 90.000,C 0.000} C_DIS
LIN {X 30.247,Y -27.308,Z -45.006,A -90.000,B 90.000,C 0.000} C_DIS
LIN {X 30.342,Y -27.308,Z -44.979,A -90.000,B 90.000,C 0.000} C_DIS
LIN {X 30.800,Y -27.308,Z -44.854,A -90.000,B 90.000,C 0.000} C_DIS
LIN {X 31.703,Y -27.308,Z -44.679,A -90.000,B 90.000,C 0.000} C_DIS
LIN {X 31.904,Y -27.308,Z -44.642,A -90.000,B 90.000,C 0.000} C_DIS
LIN {X 32.382,Y -27.308,Z -44.576,A -90.000,B 90.000,C 0.000} C_DIS
LIN {X 33.026,Y -27.308,Z -44.500,A -90.000,B 90.000,C 0.000} C_DIS
LIN {X 33.299,Y -27.308,Z -44.472,A -90.000,B 90.000,C 0.000} C_DIS
LIN {X 34.106,Y -27.308,Z -44.440,A -90.000,B 90.000,C 0.000} C_DIS
LIN {X 34.379,Y -27.308,Z -44.430,A -90.000,B 90.000,C 0.000} C_DIS
LIN {X 34.809,Y -27.308,Z -44.424,A -90.000,B 90.000,C 0.000} C_DIS
LIN {X 34.908,Y -27.308,Z -44.427,A -90.000,B 90.000,C 0.000} C_DIS
LIN {X 35.661,Y -27.308,Z -44.415,A -90.000,B 90.000,C 0.000} C_DIS
LIN {X 35.944,Y -27.308,Z -44.417,A -90.000,B 90.000,C 0.000} C_DIS
LIN {X 36.401,Y -27.308,Z -44.379,A -90.000,B 90.000,C 0.000} C_DIS
LIN {X 36.864,Y -27.308,Z -44.270,A -90.000,B 90.000,C 0.000} C_DIS
LIN {X 37.986,Y -27.308,Z -43.891,A -90.000,B 90.000,C 0.000} C_DIS
LIN {X 39.146,Y -27.308,Z -43.475,A -90.000,B 90.000,C 0.000} C_DIS
LIN {X 39.665,Y -27.308,Z -43.283,A -90.000,B 90.000,C 0.000} C_DIS
LIN {X 40.086,Y -27.308,Z -43.152,A -90.000,B 90.000,C 0.000} C_DIS
LIN {X 41.064,Y -27.308,Z -42.856,A -90.000,B 90.000,C 0.000} C_DIS
LIN {X 41.887,Y -27.308,Z -42.633,A -90.000,B 90.000,C 0.000} C_DIS
LIN {X 42.587,Y -27.308,Z -42.499,A -90.000,B 90.000,C 0.000} C_DIS
LIN {X 43.328,Y -27.308,Z -42.392,A -90.000,B 90.000,C 0.000} C_DIS
LIN {X 43.780,Y -27.308,Z -42.332,A -90.000,B 90.000,C 0.000} C_DIS
LIN {X 45.231,Y -27.308,Z -42.269,A -90.000,B 90.000,C 0.000} C_DIS
LIN {X 45.687,Y -27.308,Z -42.261,A -90.000,B 90.000,C 0.000} C_DIS
LIN {X 46.114,Y -27.308,Z -42.299,A -90.000,B 90.000,C 0.000} C_DIS
LIN {X 46.490,Y -27.308,Z -42.343,A -90.000,B 90.000,C 0.000} C_DIS
LIN {X 46.845,Y -27.308,Z -42.388,A -90.000,B 90.000,C 0.000} C_DIS
LIN {X 47.882,Y -27.308,Z -42.552,A -90.000,B 90.000,C 0.000} C_DIS
LIN {X 48.337,Y -27.308,Z -42.660,A -90.000,B 90.000,C 0.000} C_DIS
LIN {X 49.744,Y -27.308,Z -43.003,A -90.000,B 90.000,C 0.000} C_DIS
LIN {X 49.923,Y -27.308,Z -43.062,A -90.000,B 90.000,C 0.000} C_DIS
LIN {X 50.341,Y -27.308,Z -43.210,A -90.000,B 90.000,C 0.000} C_DIS
LIN {X 51.412,Y -27.308,Z -43.632,A -90.000,B 90.000,C 0.000} C_DIS
LIN {X 52.285,Y -27.308,Z -44.024,A -90.000,B 90.000,C 0.000} C_DIS
LIN {X 53.027,Y -27.308,Z -44.385,A -90.000,B 90.000,C 0.000} C_DIS
LIN {X 53.452,Y -27.308,Z -44.600,A -90.000,B 90.000,C 0.000} C_DIS
LIN {X 54.382,Y -27.308,Z -45.165,A -90.000,B 90.000,C 0.000} C_DIS
LIN {X 56.073,Y -27.308,Z -46.226,A -90.000,B 90.000,C 0.000} C_DIS
LIN {X 56.461,Y -27.308,Z -46.477,A -90.000,B 90.000,C 0.000} C_DIS
LIN {X 56.666,Y -27.308,Z -46.639,A -90.000,B 90.000,C 0.000} C_DIS
LIN {X 58.184,Y -27.308,Z -47.862,A -90.000,B 90.000,C 0.000} C_DIS
LIN {X 58.556,Y -27.308,Z -48.170,A -90.000,B 90.000,C 0.000} C_DIS
LIN {X 59.100,Y -27.308,Z -48.624,A -90.000,B 90.000,C 0.000} C_DIS
LIN {X 61.179,Y -27.308,Z -50.575,A -90.000,B 90.000,C 0.000} C_DIS
LIN {X 61.864,Y -27.308,Z -51.231,A -90.000,B 90.000,C 0.000} C_DIS
LIN {X 63.171,Y -27.308,Z -52.491,A -90.000,B 90.000,C 0.000} C_DIS
LIN {X 64.048,Y -27.308,Z -53.266,A -90.000,B 90.000,C 0.000} C_DIS
LIN {X 65.006,Y -27.308,Z -54.129,A -90.000,B 90.000,C 0.000} C_DIS
LIN {X 66.147,Y -27.308,Z -54.994,A -90.000,B 90.000,C 0.000} C_DIS
LIN {X 66.886,Y -27.308,Z -55.534,A -90.000,B 90.000,C 0.000} C_DIS
LIN {X 67.739,Y -27.308,Z -56.127,A -90.000,B 90.000,C 0.000} C_DIS
LIN {X 69.016,Y -27.308,Z -56.978,A -90.000,B 90.000,C 0.000} C_DIS
LIN {X 70.300,Y -27.308,Z -57.878,A -90.000,B 90.000,C 0.000} C_DIS
LIN {X 71.059,Y -27.308,Z -58.388,A -90.000,B 90.000,C 0.000} C_DIS
LIN {X 72.700,Y -27.308,Z -59.679,A -90.000,B 90.000,C 0.000} C_DIS
LIN {X 73.132,Y -27.308,Z -60.013,A -90.000,B 90.000,C 0.000} C_DIS
LIN {X 73.257,Y -27.308,Z -60.130,A -90.000,B 90.000,C 0.000} C_DIS
LIN {X 73.889,Y -27.308,Z -60.744,A -90.000,B 90.000,C 0.000} C_DIS
LIN {X 74.937,Y -27.308,Z -61.813,A -90.000,B 90.000,C 0.000} C_DIS
LIN {X 75.234,Y -27.308,Z -62.168,A -90.000,B 90.000,C 0.000} C_DIS
LIN {X 76.071,Y -27.308,Z -63.244,A -90.000,B 90.000,C 0.000} C_DIS
LIN {X 76.407,Y -27.308,Z -63.686,A -90.000,B 90.000,C 0.000} C_DIS
LIN {X 77.071,Y -27.308,Z -64.685,A -90.000,B 90.000,C 0.000} C_DIS
LIN {X 77.643,Y -27.308,Z -65.550,A -90.000,B 90.000,C 0.000} C_DIS
LIN {X 78.032,Y -27.308,Z -66.181,A -90.000,B 90.000,C 0.000} C_DIS
LIN {X 78.362,Y -27.308,Z -66.727,A -90.000,B 90.000,C 0.000} C_DIS
LIN {X 78.433,Y -27.308,Z -66.838,A -90.000,B 90.000,C 0.000} C_DIS
LIN {X 78.586,Y -27.308,Z -66.075,A -90.000,B 90.000,C 0.000} C_DIS
LIN {X 79.091,Y -27.308,Z -64.165,A -90.000,B 90.000,C 0.000} C_DIS
LIN {X 79.194,Y -27.308,Z -63.825,A -90.000,B 90.000,C 0.000} C_DIS
LIN {X 79.834,Y -27.308,Z -61.877,A -90.000,B 90.000,C 0.000} C_DIS
LIN {X 80.548,Y -27.308,Z -59.938,A -90.000,B 90.000,C 0.000} C_DIS
LIN {X 80.691,Y -27.308,Z -59.564,A -90.000,B 90.000,C 0.000} C_DIS
LIN {X 80.736,Y -27.308,Z -59.449,A -90.000,B 90.000,C 0.000} C_DIS
LIN {X 80.883,Y -27.308,Z -59.105,A -90.000,B 90.000,C 0.000} C_DIS
LIN {X 81.411,Y -27.308,Z -57.598,A -90.000,B 90.000,C 0.000} C_DIS
LIN {X 81.507,Y -27.308,Z -57.344,A -90.000,B 90.000,C 0.000} C_DIS
LIN {X 82.417,Y -27.308,Z -55.184,A -90.000,B 90.000,C 0.000} C_DIS
LIN {X 82.593,Y -27.308,Z -54.835,A -90.000,B 90.000,C 0.000} C_DIS
LIN {X 82.991,Y -27.308,Z -54.057,A -90.000,B 90.000,C 0.000} C_DIS
LIN {X 83.553,Y -27.308,Z -52.984,A -90.000,B 90.000,C 0.000} C_DIS
LIN {X 83.615,Y -27.308,Z -52.870,A -90.000,B 90.000,C 0.000} C_DIS
LIN {X 84.800,Y -27.308,Z -50.978,A -90.000,B 90.000,C 0.000} C_DIS
LIN {X 85.033,Y -27.308,Z -50.637,A -90.000,B 90.000,C 0.000} C_DIS
LIN {X 86.349,Y -27.308,Z -48.871,A -90.000,B 90.000,C 0.000} C_DIS
LIN {X 86.730,Y -27.308,Z -48.428,A -90.000,B 90.000,C 0.000} C_DIS
LIN {X 88.126,Y -27.308,Z -46.908,A -90.000,B 90.000,C 0.000} C_DIS
LIN {X 88.529,Y -27.308,Z -46.539,A -90.000,B 90.000,C 0.000} C_DIS
LIN {X 89.798,Y -27.308,Z -45.395,A -90.000,B 90.000,C 0.000} C_DIS
LIN {X 90.067,Y -27.308,Z -45.159,A -90.000,B 90.000,C 0.000} C_DIS
LIN {X 91.727,Y -27.308,Z -43.868,A -90.000,B 90.000,C 0.000} C_DIS
LIN {X 92.155,Y -27.308,Z -43.556,A -90.000,B 90.000,C 0.000} C_DIS
LIN {X 93.797,Y -27.308,Z -42.409,A -90.000,B 90.000,C 0.000} C_DIS
LIN {X 95.424,Y -27.308,Z -41.378,A -90.000,B 90.000,C 0.000} C_DIS
LIN {X 95.864,Y -27.308,Z -41.121,A -90.000,B 90.000,C 0.000} C_DIS
LIN {X 97.376,Y -27.308,Z -40.260,A -90.000,B 90.000,C 0.000} C_DIS
LIN {X 97.527,Y -27.308,Z -40.182,A -90.000,B 90.000,C 0.000} C_DIS
LIN {X 98.805,Y -27.308,Z -39.523,A -90.000,B 90.000,C 0.000} C_DIS
LIN {X 100.317,Y -27.308,Z -38.807,A -90.000,B 90.000,C 0.000} C_DIS
LIN {X 102.237,Y -27.308,Z -37.938,A -90.000,B 90.000,C 0.000} C_DIS
LIN {X 103.453,Y -27.308,Z -37.395,A -90.000,B 90.000,C 0.000} C_DIS
LIN {X 104.516,Y -27.308,Z -36.925,A -90.000,B 90.000,C 0.000} C_DIS
LIN {X 105.407,Y -27.308,Z -36.550,A -90.000,B 90.000,C 0.000} C_DIS
LIN {X 106.871,Y -27.308,Z -35.969,A -90.000,B 90.000,C 0.000} C_DIS
LIN {X 107.396,Y -27.308,Z -35.770,A -90.000,B 90.000,C 0.000} C_DIS
LIN {X 107.855,Y -27.308,Z -35.604,A -90.000,B 90.000,C 0.000} C_DIS
LIN {X 108.317,Y -27.308,Z -35.448,A -90.000,B 90.000,C 0.000} C_DIS
LIN {X 108.770,Y -27.308,Z -35.327,A -90.000,B 90.000,C 0.000} C_DIS
LIN {X 109.221,Y -27.308,Z -35.225,A -90.000,B 90.000,C 0.000} C_DIS
LIN {X 109.732,Y -27.308,Z -35.159,A -90.000,B 90.000,C 0.000} C_DIS
LIN {X 110.108,Y -27.308,Z -35.113,A -90.000,B 90.000,C 0.000} C_DIS
LIN {X 110.615,Y -27.308,Z -35.106,A -90.000,B 90.000,C 0.000} C_DIS
LIN {X 110.949,Y -27.308,Z -35.117,A -90.000,B 90.000,C 0.000} C_DIS
LIN {X 111.443,Y -27.308,Z -35.160,A -90.000,B 90.000,C 0.000} C_DIS
LIN {X 112.087,Y -27.308,Z -35.282,A -90.000,B 90.000,C 0.000} C_DIS
LIN {X 112.431,Y -27.308,Z -35.370,A -90.000,B 90.000,C 0.000} C_DIS
LIN {X 112.915,Y -27.308,Z -35.515,A -90.000,B 90.000,C 0.000} C_DIS
LIN {X 113.055,Y -27.308,Z -35.560,A -90.000,B 90.000,C 0.000} C_DIS
LIN {X 113.505,Y -27.308,Z -35.746,A -90.000,B 90.000,C 0.000} C_DIS
LIN {X 113.979,Y -27.308,Z -35.973,A -90.000,B 90.000,C 0.000} C_DIS
LIN {X 114.416,Y -27.308,Z -36.209,A -90.000,B 90.000,C 0.000} C_DIS
LIN {X 114.565,Y -27.308,Z -36.302,A -90.000,B 90.000,C 0.000} C_DIS
LIN {X 114.950,Y -27.308,Z -36.565,A -90.000,B 90.000,C 0.000} C_DIS
LIN {X 115.050,Y -27.308,Z -36.644,A -90.000,B 90.000,C 0.000} C_DIS
LIN {X 115.445,Y -27.308,Z -36.978,A -90.000,B 90.000,C 0.000} C_DIS
LIN {X 115.513,Y -27.308,Z -37.039,A -90.000,B 90.000,C 0.000} C_DIS
LIN {X 115.852,Y -27.308,Z -37.389,A -90.000,B 90.000,C 0.000} C_DIS
LIN {X 116.079,Y -27.308,Z -37.631,A -90.000,B 90.000,C 0.000} C_DIS
LIN {X 116.439,Y -27.308,Z -38.088,A -90.000,B 90.000,C 0.000} C_DIS
LIN {X 116.700,Y -27.308,Z -38.500,A -90.000,B 90.000,C 0.000} C_DIS
LIN {X 116.926,Y -27.308,Z -38.957,A -90.000,B 90.000,C 0.000} C_DIS
LIN {X 117.065,Y -27.308,Z -39.264,A -90.000,B 90.000,C 0.000} C_DIS
LIN {X 117.133,Y -27.308,Z -39.442,A -90.000,B 90.000,C 0.000} C_DIS
LIN {X 117.260,Y -27.308,Z -39.781,A -90.000,B 90.000,C 0.000} C_DIS
LIN {X 117.389,Y -27.308,Z -40.275,A -90.000,B 90.000,C 0.000} C_DIS
LIN {X 117.462,Y -27.308,Z -40.593,A -90.000,B 90.000,C 0.000} C_DIS
LIN {X 117.540,Y -27.308,Z -41.102,A -90.000,B 90.000,C 0.000} C_DIS
LIN {X 117.595,Y -27.308,Z -41.518,A -90.000,B 90.000,C 0.000} C_DIS
LIN {X 117.630,Y -27.308,Z -41.874,A -90.000,B 90.000,C 0.000} C_DIS
LIN {X 117.658,Y -27.308,Z -42.443,A -90.000,B 90.000,C 0.000} C_DIS
LIN {X 117.668,Y -27.308,Z -42.694,A -90.000,B 90.000,C 0.000} C_DIS
LIN {X 117.662,Y -27.308,Z -42.930,A -90.000,B 90.000,C 0.000} C_DIS
LIN {X 117.651,Y -27.308,Z -43.202,A -90.000,B 90.000,C 0.000} C_DIS
LIN {X 117.608,Y -27.308,Z -43.715,A -90.000,B 90.000,C 0.000} C_DIS
LIN {X 117.567,Y -27.308,Z -44.117,A -90.000,B 90.000,C 0.000} C_DIS
LIN {X 117.484,Y -27.308,Z -44.664,A -90.000,B 90.000,C 0.000} C_DIS
LIN {X 117.391,Y -27.308,Z -45.152,A -90.000,B 90.000,C 0.000} C_DIS
LIN {X 117.260,Y -27.308,Z -45.739,A -90.000,B 90.000,C 0.000} C_DIS
LIN {X 117.108,Y -27.308,Z -46.251,A -90.000,B 90.000,C 0.000} C_DIS
LIN {X 116.900,Y -27.308,Z -46.938,A -90.000,B 90.000,C 0.000} C_DIS
LIN {X 116.548,Y -27.308,Z -47.851,A -90.000,B 90.000,C 0.000} C_DIS
LIN {X 116.372,Y -27.308,Z -48.278,A -90.000,B 90.000,C 0.000} C_DIS
LIN {X 115.873,Y -27.308,Z -49.350,A -90.000,B 90.000,C 0.000} C_DIS
LIN {X 115.132,Y -27.308,Z -50.830,A -90.000,B 90.000,C 0.000} C_DIS
LIN {X 114.586,Y -27.308,Z -51.912,A -90.000,B 90.000,C 0.000} C_DIS
LIN {X 113.941,Y -27.308,Z -53.229,A -90.000,B 90.000,C 0.000} C_DIS
LIN {X 113.276,Y -27.308,Z -54.687,A -90.000,B 90.000,C 0.000} C_DIS
LIN {X 112.799,Y -27.308,Z -55.830,A -90.000,B 90.000,C 0.000} C_DIS
LIN {X 112.213,Y -27.308,Z -57.388,A -90.000,B 90.000,C 0.000} C_DIS
LIN {X 111.674,Y -27.308,Z -59.009,A -90.000,B 90.000,C 0.000} C_DIS
LIN {X 111.236,Y -27.308,Z -60.534,A -90.000,B 90.000,C 0.000} C_DIS
LIN {X 110.710,Y -27.308,Z -62.458,A -90.000,B 90.000,C 0.000} C_DIS
LIN {X 110.135,Y -27.308,Z -64.496,A -90.000,B 90.000,C 0.000} C_DIS
LIN {X 109.994,Y -27.308,Z -64.968,A -90.000,B 90.000,C 0.000} C_DIS
LIN {X 109.345,Y -27.308,Z -67.050,A -90.000,B 90.000,C 0.000} C_DIS
LIN {X 108.519,Y -27.308,Z -69.358,A -90.000,B 90.000,C 0.000} C_DIS
LIN {X 107.562,Y -27.308,Z -71.765,A -90.000,B 90.000,C 0.000} C_DIS
LIN {X 107.403,Y -27.308,Z -72.150,A -90.000,B 90.000,C 0.000} C_DIS
LIN {X 106.414,Y -27.308,Z -74.420,A -90.000,B 90.000,C 0.000} C_DIS
LIN {X 105.411,Y -27.308,Z -76.516,A -90.000,B 90.000,C 0.000} C_DIS
LIN {X 104.209,Y -27.308,Z -78.763,A -90.000,B 90.000,C 0.000} C_DIS
LIN {X 103.956,Y -27.308,Z -79.201,A -90.000,B 90.000,C 0.000} C_DIS
LIN {X 103.058,Y -27.308,Z -80.726,A -90.000,B 90.000,C 0.000} C_DIS
LIN {X 102.174,Y -27.308,Z -82.113,A -90.000,B 90.000,C 0.000} C_DIS
LIN {X 99.671,Y -27.308,Z -85.862,A -90.000,B 90.000,C 0.000} C_DIS
LIN {X 99.672,Y -27.308,Z -86.054,A -90.000,B 90.000,C 0.000} C_DIS
LIN {X 99.706,Y -27.308,Z -86.876,A -90.000,B 90.000,C 0.000} C_DIS
LIN {X 99.730,Y -27.308,Z -87.350,A -90.000,B 90.000,C 0.000} C_DIS
LIN {X 99.760,Y -27.308,Z -89.238,A -90.000,B 90.000,C 0.000} C_DIS
LIN {X 99.804,Y -27.308,Z -90.574,A -90.000,B 90.000,C 0.000} C_DIS
LIN {X 99.802,Y -27.308,Z -90.723,A -90.000,B 90.000,C 0.000} C_DIS
LIN {X 99.766,Y -27.308,Z -92.076,A -90.000,B 90.000,C 0.000} C_DIS
LIN {X 99.744,Y -27.308,Z -92.713,A -90.000,B 90.000,C 0.000} C_DIS
LIN {X 99.703,Y -27.308,Z -93.440,A -90.000,B 90.000,C 0.000} C_DIS
LIN {X 99.624,Y -27.308,Z -94.093,A -90.000,B 90.000,C 0.000} C_DIS
LIN {X 99.441,Y -27.308,Z -95.339,A -90.000,B 90.000,C 0.000} C_DIS
LIN {X 99.378,Y -27.308,Z -95.847,A -90.000,B 90.000,C 0.000} C_DIS
LIN {X 99.108,Y -27.308,Z -97.279,A -90.000,B 90.000,C 0.000} C_DIS
LIN {X 99.074,Y -27.308,Z -97.824,A -90.000,B 90.000,C 0.000} C_DIS
LIN {X 99.067,Y -27.308,Z -97.935,A -90.000,B 90.000,C 0.000} C_DIS
LIN {X 98.999,Y -27.308,Z -98.406,A -90.000,B 90.000,C 0.000} C_DIS
LIN {X 98.847,Y -27.308,Z -99.372,A -90.000,B 90.000,C 0.000} C_DIS
LIN {X 98.832,Y -27.308,Z -99.587,A -90.000,B 90.000,C 0.000} C_DIS
LIN {X 98.643,Y -27.308,Z -101.062,A -90.000,B 90.000,C 0.000} C_DIS
LIN {X 98.635,Y -27.308,Z -101.244,A -90.000,B 90.000,C 0.000} C_DIS
LIN {X 98.514,Y -27.308,Z -102.485,A -90.000,B 90.000,C 0.000} C_DIS
LIN {X 98.487,Y -27.308,Z -102.724,A -90.000,B 90.000,C 0.000} C_DIS
LIN {X 98.410,Y -27.308,Z -104.002,A -90.000,B 90.000,C 0.000} C_DIS
LIN {X 98.416,Y -27.308,Z -104.245,A -90.000,B 90.000,C 0.000} C_DIS
LIN {X 98.436,Y -27.308,Z -104.793,A -90.000,B 90.000,C 0.000} C_DIS
LIN {X 98.553,Y -27.308,Z -105.741,A -90.000,B 90.000,C 0.000} C_DIS
LIN {X 98.742,Y -27.308,Z -106.868,A -90.000,B 90.000,C 0.000} C_DIS
LIN {X 98.927,Y -27.308,Z -108.071,A -90.000,B 90.000,C 0.000} C_DIS
LIN {X 98.995,Y -27.308,Z -108.826,A -90.000,B 90.000,C 0.000} C_DIS
LIN {X 99.065,Y -27.308,Z -109.529,A -90.000,B 90.000,C 0.000} C_DIS
LIN {X 99.124,Y -27.308,Z -110.547,A -90.000,B 90.000,C 0.000} C_DIS
LIN {X 99.170,Y -27.308,Z -111.220,A -90.000,B 90.000,C 0.000} C_DIS
LIN {X 99.195,Y -27.308,Z -111.675,A -90.000,B 90.000,C 0.000} C_DIS
LIN {X 99.250,Y -27.308,Z -112.941,A -90.000,B 90.000,C 0.000} C_DIS
LIN {X 99.285,Y -27.308,Z -113.571,A -90.000,B 90.000,C 0.000} C_DIS
LIN {X 99.356,Y -27.308,Z -115.258,A -90.000,B 90.000,C 0.000} C_DIS
LIN {X 99.402,Y -27.308,Z -116.060,A -90.000,B 90.000,C 0.000} C_DIS
LIN {X 99.483,Y -27.308,Z -117.765,A -90.000,B 90.000,C 0.000} C_DIS
LIN {X 99.501,Y -27.308,Z -118.095,A -90.000,B 90.000,C 0.000} C_DIS
LIN {X 99.596,Y -27.308,Z -120.195,A -90.000,B 90.000,C 0.000} C_DIS
LIN {X 99.668,Y -27.308,Z -122.369,A -90.000,B 90.000,C 0.000} C_DIS
LIN {X 99.672,Y -27.308,Z -122.494,A -90.000,B 90.000,C 0.000} C_DIS
LIN {X 99.705,Y -27.308,Z -124.859,A -90.000,B 90.000,C 0.000} C_DIS
LIN {X 99.674,Y -27.308,Z -127.095,A -90.000,B 90.000,C 0.000} C_DIS
LIN {X 99.669,Y -27.308,Z -127.298,A -90.000,B 90.000,C 0.000} C_DIS
LIN {X 99.576,Y -27.308,Z -129.602,A -90.000,B 90.000,C 0.000} C_DIS
LIN {X 99.430,Y -27.308,Z -132.093,A -90.000,B 90.000,C 0.000} C_DIS
LIN {X 99.401,Y -27.308,Z -132.491,A -90.000,B 90.000,C 0.000} C_DIS
LIN {X 99.240,Y -27.308,Z -134.869,A -90.000,B 90.000,C 0.000} C_DIS
LIN {X 99.055,Y -27.308,Z -137.496,A -90.000,B 90.000,C 0.000} C_DIS
LIN {X 99.014,Y -27.308,Z -138.047,A -90.000,B 90.000,C 0.000} C_DIS
LIN {X 98.786,Y -27.308,Z -140.976,A -90.000,B 90.000,C 0.000} C_DIS
LIN {X 98.742,Y -27.308,Z -141.512,A -90.000,B 90.000,C 0.000} C_DIS
LIN {X 98.453,Y -27.308,Z -144.726,A -90.000,B 90.000,C 0.000} C_DIS
LIN {X 98.409,Y -27.308,Z -145.194,A -90.000,B 90.000,C 0.000} C_DIS
LIN {X 98.000,Y -27.308,Z -149.032,A -90.000,B 90.000,C 0.000} C_DIS
LIN {X 97.974,Y -27.308,Z -149.268,A -90.000,B 90.000,C 0.000} C_DIS
LIN {X 97.503,Y -27.308,Z -152.892,A -90.000,B 90.000,C 0.000} C_DIS
LIN {X 97.368,Y -27.308,Z -153.883,A -90.000,B 90.000,C 0.000} C_DIS
LIN {X 96.787,Y -27.308,Z -157.725,A -90.000,B 90.000,C 0.000} C_DIS
LIN {X 96.371,Y -27.308,Z -160.130,A -90.000,B 90.000,C 0.000} C_DIS
LIN {X 96.129,Y -27.308,Z -161.572,A -90.000,B 90.000,C 0.000} C_DIS
LIN {X 95.887,Y -27.308,Z -162.842,A -90.000,B 90.000,C 0.000} C_DIS
LIN {X 95.656,Y -27.308,Z -164.042,A -90.000,B 90.000,C 0.000} C_DIS
LIN {X 95.157,Y -27.308,Z -166.756,A -90.000,B 90.000,C 0.000} C_DIS
LIN {X 94.964,Y -27.308,Z -167.662,A -90.000,B 90.000,C 0.000} C_DIS
LIN {X 94.382,Y -27.308,Z -170.650,A -90.000,B 90.000,C 0.000} C_DIS
LIN {X 94.253,Y -27.308,Z -171.220,A -90.000,B 90.000,C 0.000} C_DIS
LIN {X 94.233,Y -27.308,Z -171.347,A -90.000,B 90.000,C 0.000} C_DIS
LIN {X 93.664,Y -27.308,Z -174.251,A -90.000,B 90.000,C 0.000} C_DIS
LIN {X 93.593,Y -27.308,Z -174.722,A -90.000,B 90.000,C 0.000} C_DIS
LIN {X 93.562,Y -27.308,Z -174.892,A -90.000,B 90.000,C 0.000} C_DIS
LIN {X 93.252,Y -27.308,Z -176.513,A -90.000,B 90.000,C 0.000} C_DIS
LIN {X 93.035,Y -27.308,Z -178.012,A -90.000,B 90.000,C 0.000} C_DIS
LIN {X 92.825,Y -27.308,Z -179.216,A -90.000,B 90.000,C 0.000} C_DIS
LIN {X 92.607,Y -27.308,Z -180.948,A -90.000,B 90.000,C 0.000} C_DIS
LIN {X 92.501,Y -27.308,Z -181.650,A -90.000,B 90.000,C 0.000} C_DIS
LIN {X 92.309,Y -27.308,Z -183.524,A -90.000,B 90.000,C 0.000} C_DIS
LIN {X 92.225,Y -27.308,Z -184.538,A -90.000,B 90.000,C 0.000} C_DIS
LIN {X 92.131,Y -27.308,Z -185.560,A -90.000,B 90.000,C 0.000} C_DIS
LIN {X 92.118,Y -27.308,Z -185.774,A -90.000,B 90.000,C 0.000} C_DIS
LIN {X 91.991,Y -27.308,Z -187.551,A -90.000,B 90.000,C 0.000} C_DIS
LIN {X 91.960,Y -27.308,Z -188.214,A -90.000,B 90.000,C 0.000} C_DIS
LIN {X 91.909,Y -27.308,Z -189.153,A -90.000,B 90.000,C 0.000} C_DIS
LIN {X 91.865,Y -27.308,Z -190.490,A -90.000,B 90.000,C 0.000} C_DIS
LIN {X 91.861,Y -27.308,Z -190.611,A -90.000,B 90.000,C 0.000} C_DIS
LIN {X 91.827,Y -27.308,Z -191.124,A -90.000,B 90.000,C 0.000} C_DIS
LIN {X 91.723,Y -27.308,Z -193.200,A -90.000,B 90.000,C 0.000} C_DIS
LIN {X 91.695,Y -27.308,Z -193.506,A -90.000,B 90.000,C 0.000} C_DIS
LIN {X 91.405,Y -27.308,Z -196.490,A -90.000,B 90.000,C 0.000} C_DIS
LIN {X 91.359,Y -27.308,Z -196.807,A -90.000,B 90.000,C 0.000} C_DIS
LIN {X 90.822,Y -27.308,Z -199.954,A -90.000,B 90.000,C 0.000} C_DIS
LIN {X 90.790,Y -27.308,Z -200.114,A -90.000,B 90.000,C 0.000} C_DIS
LIN {X 89.886,Y -27.308,Z -204.324,A -90.000,B 90.000,C 0.000} C_DIS
LIN {X 88.760,Y -27.308,Z -209.050,A -90.000,B 90.000,C 0.000} C_DIS
LIN {X 88.010,Y -27.308,Z -212.061,A -90.000,B 90.000,C 0.000} C_DIS
LIN {X 87.487,Y -27.308,Z -214.179,A -90.000,B 90.000,C 0.000} C_DIS
LIN {X 86.889,Y -27.308,Z -216.558,A -90.000,B 90.000,C 0.000} C_DIS
LIN {X 85.924,Y -27.308,Z -220.488,A -90.000,B 90.000,C 0.000} C_DIS
LIN {X 84.901,Y -27.308,Z -224.831,A -90.000,B 90.000,C 0.000} C_DIS
LIN {X 84.678,Y -27.308,Z -225.734,A -90.000,B 90.000,C 0.000} C_DIS
LIN {X 83.482,Y -27.308,Z -230.535,A -90.000,B 90.000,C 0.000} C_DIS
LIN {X 83.339,Y -27.308,Z -231.042,A -90.000,B 90.000,C 0.000} C_DIS
LIN {X 81.710,Y -27.308,Z -236.616,A -90.000,B 90.000,C 0.000} C_DIS
LIN {X 80.664,Y -27.308,Z -239.719,A -90.000,B 90.000,C 0.000} C_DIS
LIN {X 79.774,Y -27.308,Z -242.345,A -90.000,B 90.000,C 0.000} C_DIS
LIN {X 79.674,Y -27.308,Z -242.644,A -90.000,B 90.000,C 0.000} C_DIS
LIN {X 79.313,Y -27.308,Z -243.561,A -90.000,B 90.000,C 0.000} C_DIS
LIN {X 79.313,Y -60.000,Z -243.561,A -90.000,B 90.000,C 0.000} C_DIS
LIN {X 99.737,Y -60.000,Z -85.762,A -90.000,B 90.000,C 0.000} C_DIS
LIN {X 99.737,Y -25.308,Z -85.762,A -90.000,B 90.000,C 0.000} C_DIS
LIN {X 99.743,Y -25.309,Z -85.835,A -90.000,B 90.000,C 0.000} C_DIS
LIN {X 99.776,Y -25.311,Z -86.266,A -90.000,B 90.000,C 0.000} C_DIS
LIN {X 99.848,Y -25.312,Z -87.594,A -90.000,B 90.000,C 0.000} C_DIS
LIN {X 99.950,Y -25.318,Z -88.761,A -90.000,B 90.000,C 0.000} C_DIS
LIN {X 99.975,Y -25.320,Z -89.231,A -90.000,B 90.000,C 0.000} C_DIS
LIN {X 99.996,Y -25.320,Z -89.787,A -90.000,B 90.000,C 0.000} C_DIS
LIN {X 100.011,Y -25.319,Z -90.575,A -90.000,B 90.000,C 0.000} C_DIS
LIN {X 100.027,Y -25.324,Z -91.607,A -90.000,B 90.000,C 0.000} C_DIS
LIN {X 100.040,Y -25.327,Z -92.070,A -90.000,B 90.000,C 0.000} C_DIS
LIN {X 100.040,Y -25.327,Z -92.120,A -90.000,B 90.000,C 0.000} C_DIS
LIN {X 99.989,Y -25.325,Z -92.994,A -90.000,B 90.000,C 0.000} C_DIS
LIN {X 99.970,Y -25.327,Z -93.472,A -90.000,B 90.000,C 0.000} C_DIS
LIN {X 99.951,Y -25.332,Z -93.951,A -90.000,B 90.000,C 0.000} C_DIS
LIN {X 99.929,Y -25.337,Z -94.355,A -90.000,B 90.000,C 0.000} C_DIS
LIN {X 99.903,Y -25.338,Z -94.572,A -90.000,B 90.000,C 0.000} C_DIS
LIN {X 99.811,Y -25.344,Z -95.418,A -90.000,B 90.000,C 0.000} C_DIS
LIN {X 99.790,Y -25.352,Z -95.911,A -90.000,B 90.000,C 0.000} C_DIS
LIN {X 99.734,Y -25.359,Z -96.366,A -90.000,B 90.000,C 0.000} C_DIS
LIN {X 99.681,Y -25.360,Z -96.671,A -90.000,B 90.000,C 0.000} C_DIS
LIN {X 99.640,Y -25.381,Z -97.332,A -90.000,B 90.000,C 0.000} C_DIS
LIN {X 99.631,Y -25.381,Z -97.497,A -90.000,B 90.000,C 0.000} C_DIS
LIN {X 99.602,Y -25.381,Z -97.965,A -90.000,B 90.000,C 0.000} C_DIS
LIN {X 99.588,Y -25.385,Z -98.162,A -90.000,B 90.000,C 0.000} C_DIS
LIN {X 99.522,Y -25.408,Z -99.100,A -90.000,B 90.000,C 0.000} C_DIS
LIN {X 99.492,Y -25.409,Z -99.312,A -90.000,B 90.000,C 0.000} C_DIS
LIN {X 99.482,Y -25.413,Z -99.443,A -90.000,B 90.000,C 0.000} C_DIS
LIN {X 99.471,Y -25.413,Z -99.607,A -90.000,B 90.000,C 0.000} C_DIS
LIN {X 99.397,Y -25.432,Z -100.628,A -90.000,B 90.000,C 0.000} C_DIS
LIN {X 99.351,Y -25.432,Z -100.989,A -90.000,B 90.000,C 0.000} C_DIS
LIN {X 99.345,Y -25.436,Z -101.105,A -90.000,B 90.000,C 0.000} C_DIS
LIN {X 99.338,Y -25.436,Z -101.270,A -90.000,B 90.000,C 0.000} C_DIS
LIN {X 99.290,Y -25.453,Z -102.243,A -90.000,B 90.000,C 0.000} C_DIS
LIN {X 99.268,Y -25.453,Z -102.477,A -90.000,B 90.000,C 0.000} C_DIS
LIN {X 99.261,Y -25.466,Z -102.814,A -90.000,B 90.000,C 0.000} C_DIS
LIN {X 99.256,Y -25.475,Z -103.262,A -90.000,B 90.000,C 0.000} C_DIS
LIN {X 99.232,Y -25.479,Z -103.803,A -90.000,B 90.000,C 0.000} C_DIS
LIN {X 99.238,Y -25.487,Z -103.991,A -90.000,B 90.000,C 0.000} C_DIS
LIN {X 99.275,Y -25.496,Z -104.576,A -90.000,B 90.000,C 0.000} C_DIS
LIN {X 99.293,Y -25.502,Z -104.735,A -90.000,B 90.000,C 0.000} C_DIS
LIN {X 99.345,Y -25.503,Z -105.137,A -90.000,B 90.000,C 0.000} C_DIS
LIN {X 99.398,Y -25.505,Z -105.521,A -90.000,B 90.000,C 0.000} C_DIS
LIN {X 99.418,Y -25.508,Z -105.639,A -90.000,B 90.000,C 0.000} C_DIS
LIN {X 99.538,Y -25.509,Z -106.332,A -90.000,B 90.000,C 0.000} C_DIS
LIN {X 99.584,Y -25.509,Z -106.611,A -90.000,B 90.000,C 0.000} C_DIS
LIN {X 99.804,Y -25.512,Z -108.003,A -90.000,B 90.000,C 0.000} C_DIS
LIN {X 99.889,Y -25.516,Z -108.848,A -90.000,B 90.000,C 0.000} C_DIS
LIN {X 99.954,Y -25.518,Z -109.453,A -90.000,B 90.000,C 0.000} C_DIS
LIN {X 100.042,Y -25.525,Z -110.714,A -90.000,B 90.000,C 0.000} C_DIS
LIN {X 100.076,Y -25.528,Z -111.124,A -90.000,B 90.000,C 0.000} C_DIS
LIN {X 100.094,Y -25.528,Z -111.435,A -90.000,B 90.000,C 0.000} C_DIS
LIN {X 100.138,Y -25.532,Z -112.210,A -90.000,B 90.000,C 0.000} C_DIS
LIN {X 100.185,Y -25.541,Z -112.896,A -90.000,B 90.000,C 0.000} C_DIS
LIN {X 100.222,Y -25.542,Z -113.532,A -90.000,B 90.000,C 0.000} C_DIS
LIN {X 100.255,Y -25.545,Z -114.157,A -90.000,B 90.000,C 0.000} C_DIS
LIN {X 100.312,Y -25.557,Z -115.040,A -90.000,B 90.000,C 0.000} C_DIS
LIN {X 100.367,Y -25.564,Z -115.782,A -90.000,B 90.000,C 0.000} C_DIS
LIN {X 100.452,Y -25.572,Z -117.264,A -90.000,B 90.000,C 0.000} C_DIS
LIN {X 100.491,Y -25.578,Z -117.822,A -90.000,B 90.000,C 0.000} C_DIS
LIN {X 100.566,Y -25.584,Z -119.212,A -90.000,B 90.000,C 0.000} C_DIS
LIN {X 100.606,Y -25.589,Z -119.931,A -90.000,B 90.000,C 0.000} C_DIS
LIN {X 100.626,Y -25.591,Z -120.320,A -90.000,B 90.000,C 0.000} C_DIS
LIN {X 100.715,Y -25.602,Z -122.450,A -90.000,B 90.000,C 0.000} C_DIS
LIN {X 100.735,Y -25.609,Z -123.080,A -90.000,B 90.000,C 0.000} C_DIS
LIN {X 100.772,Y -25.617,Z -124.807,A -90.000,B 90.000,C 0.000} C_DIS
LIN {X 100.759,Y -25.626,Z -126.808,A -90.000,B 90.000,C 0.000} C_DIS
LIN {X 100.760,Y -25.629,Z -127.109,A -90.000,B 90.000,C 0.000} C_DIS
LIN {X 100.756,Y -25.629,Z -127.293,A -90.000,B 90.000,C 0.000} C_DIS
LIN {X 100.677,Y -25.640,Z -129.680,A -90.000,B 90.000,C 0.000} C_DIS
LIN {X 100.547,Y -25.650,Z -132.159,A -90.000,B 90.000,C 0.000} C_DIS
LIN {X 100.370,Y -25.660,Z -134.949,A -90.000,B 90.000,C 0.000} C_DIS
LIN {X 100.170,Y -25.667,Z -137.917,A -90.000,B 90.000,C 0.000} C_DIS
LIN {X 99.898,Y -25.676,Z -141.556,A -90.000,B 90.000,C 0.000} C_DIS
LIN {X 99.829,Y -25.679,Z -142.382,A -90.000,B 90.000,C 0.000} C_DIS
LIN {X 99.595,Y -25.690,Z -145.140,A -90.000,B 90.000,C 0.000} C_DIS
LIN {X 99.435,Y -25.706,Z -146.865,A -90.000,B 90.000,C 0.000} C_DIS
LIN {X 99.189,Y -25.720,Z -149.332,A -90.000,B 90.000,C 0.000} C_DIS
LIN {X 99.130,Y -25.723,Z -149.830,A -90.000,B 90.000,C 0.000} C_DIS
LIN {X 98.944,Y -25.734,Z -151.378,A -90.000,B 90.000,C 0.000} C_DIS
LIN {X 98.766,Y -25.758,Z -152.981,A -90.000,B 90.000,C 0.000} C_DIS
LIN {X 98.623,Y -25.760,Z -154.054,A -90.000,B 90.000,C 0.000} C_DIS
LIN {X 98.502,Y -25.768,Z -154.920,A -90.000,B 90.000,C 0.000} C_DIS
LIN {X 98.285,Y -25.801,Z -156.615,A -90.000,B 90.000,C 0.000} C_DIS
LIN {X 98.098,Y -25.803,Z -157.865,A -90.000,B 90.000,C 0.000} C_DIS
LIN {X 97.780,Y -25.856,Z -160.054,A -90.000,B 90.000,C 0.000} C_DIS
LIN {X 97.720,Y -25.861,Z -160.437,A -90.000,B 90.000,C 0.000} C_DIS
LIN {X 97.635,Y -25.862,Z -160.947,A -90.000,B 90.000,C 0.000} C_DIS
LIN {X 97.506,Y -25.876,Z -161.803,A -90.000,B 90.000,C 0.000} C_DIS
LIN {X 97.198,Y -25.930,Z -163.693,A -90.000,B 90.000,C 0.000} C_DIS
LIN {X 97.133,Y -25.939,Z -164.073,A -90.000,B 90.000,C 0.000} C_DIS
LIN {X 97.050,Y -25.941,Z -164.534,A -90.000,B 90.000,C 0.000} C_DIS
LIN {X 96.639,Y -25.987,Z -166.995,A -90.000,B 90.000,C 0.000} C_DIS
LIN {X 96.584,Y -25.997,Z -167.296,A -90.000,B 90.000,C 0.000} C_DIS
LIN {X 96.553,Y -26.006,Z -167.483,A -90.000,B 90.000,C 0.000} C_DIS
LIN {X 96.482,Y -26.017,Z -167.861,A -90.000,B 90.000,C 0.000} C_DIS
LIN {X 96.013,Y -26.069,Z -170.487,A -90.000,B 90.000,C 0.000} C_DIS
LIN {X 95.939,Y -26.086,Z -170.937,A -90.000,B 90.000,C 0.000} C_DIS
LIN {X 95.903,Y -26.096,Z -171.130,A -90.000,B 90.000,C 0.000} C_DIS
LIN {X 95.826,Y -26.109,Z -171.518,A -90.000,B 90.000,C 0.000} C_DIS
LIN {X 95.818,Y -26.109,Z -171.570,A -90.000,B 90.000,C 0.000} C_DIS
LIN {X 95.377,Y -26.155,Z -174.008,A -90.000,B 90.000,C 0.000} C_DIS
LIN {X 95.288,Y -26.176,Z -174.537,A -90.000,B 90.000,C 0.000} C_DIS
LIN {X 95.270,Y -26.178,Z -174.663,A -90.000,B 90.000,C 0.000} C_DIS
LIN {X 95.224,Y -26.178,Z -174.969,A -90.000,B 90.000,C 0.000} C_DIS
LIN {X 95.195,Y -26.180,Z -175.145,A -90.000,B 90.000,C 0.000} C_DIS
LIN {X 94.945,Y -26.207,Z -176.543,A -90.000,B 90.000,C 0.000} C_DIS
LIN {X 94.904,Y -26.216,Z -176.790,A -90.000,B 90.000,C 0.000} C_DIS
LIN {X 94.728,Y -26.238,Z -178.114,A -90.000,B 90.000,C 0.000} C_DIS
LIN {X 94.708,Y -26.239,Z -178.254,A -90.000,B 90.000,C 0.000} C_DIS
LIN {X 94.534,Y -26.258,Z -179.322,A -90.000,B 90.000,C 0.000} C_DIS
LIN {X 94.512,Y -26.263,Z -179.469,A -90.000,B 90.000,C 0.000} C_DIS
LIN {X 94.405,Y -26.275,Z -180.381,A -90.000,B 90.000,C 0.000} C_DIS
LIN {X 94.310,Y -26.285,Z -181.173,A -90.000,B 90.000,C 0.000} C_DIS
LIN {X 94.245,Y -26.292,Z -181.634,A -90.000,B 90.000,C 0.000} C_DIS
LIN {X 94.214,Y -26.299,Z -181.867,A -90.000,B 90.000,C 0.000} C_DIS
LIN {X 94.108,Y -26.311,Z -182.975,A -90.000,B 90.000,C 0.000} C_DIS
LIN {X 94.040,Y -26.316,Z -183.667,A -90.000,B 90.000,C 0.000} C_DIS
LIN {X 93.963,Y -26.324,Z -184.648,A -90.000,B 90.000,C 0.000} C_DIS
LIN {X 93.876,Y -26.337,Z -185.679,A -90.000,B 90.000,C 0.000} C_DIS
LIN {X 93.864,Y -26.335,Z -185.837,A -90.000,B 90.000,C 0.000} C_DIS
LIN {X 93.731,Y -26.326,Z -187.646,A -90.000,B 90.000,C 0.000} C_DIS
LIN {X 93.696,Y -26.316,Z -188.269,A -90.000,B 90.000,C 0.000} C_DIS
LIN {X 93.640,Y -26.308,Z -189.209,A -90.000,B 90.000,C 0.000} C_DIS
LIN {X 93.614,Y -26.297,Z -189.783,A -90.000,B 90.000,C 0.000} C_DIS
LIN {X 93.578,Y -26.283,Z -190.666,A -90.000,B 90.000,C 0.000} C_DIS
LIN {X 93.539,Y -26.277,Z -191.210,A -90.000,B 90.000,C 0.000} C_DIS
LIN {X 93.413,Y -26.241,Z -193.284,A -90.000,B 90.000,C 0.000} C_DIS
LIN {X 93.388,Y -26.240,Z -193.558,A -90.000,B 90.000,C 0.000} C_DIS
LIN {X 93.081,Y -26.201,Z -196.471,A -90.000,B 90.000,C 0.000} C_DIS
LIN {X 93.053,Y -26.195,Z -196.694,A -90.000,B 90.000,C 0.000} C_DIS
LIN {X 92.990,Y -26.190,Z -197.108,A -90.000,B 90.000,C 0.000} C_DIS
LIN {X 92.498,Y -26.188,Z -199.978,A -90.000,B 90.000,C 0.000} C_DIS
LIN {X 92.464,Y -26.185,Z -200.170,A -90.000,B 90.000,C 0.000} C_DIS
LIN {X 92.428,Y -26.183,Z -200.357,A -90.000,B 90.000,C 0.000} C_DIS
LIN {X 91.596,Y -26.180,Z -204.224,A -90.000,B 90.000,C 0.000} C_DIS
LIN {X 91.500,Y -26.177,Z -204.663,A -90.000,B 90.000,C 0.000} C_DIS
LIN {X 91.338,Y -26.177,Z -205.344,A -90.000,B 90.000,C 0.000} C_DIS
LIN {X 90.346,Y -26.150,Z -209.428,A -90.000,B 90.000,C 0.000} C_DIS
LIN {X 89.732,Y -26.138,Z -211.860,A -90.000,B 90.000,C 0.000} C_DIS
LIN {X 89.184,Y -26.119,Z -214.012,A -90.000,B 90.000,C 0.000} C_DIS
LIN {X 89.098,Y -26.117,Z -214.358,A -90.000,B 90.000,C 0.000} C_DIS
LIN {X 88.436,Y -26.100,Z -216.943,A -90.000,B 90.000,C 0.000} C_DIS
LIN {X 88.002,Y -26.084,Z -218.657,A -90.000,B 90.000,C 0.000} C_DIS
LIN {X 87.455,Y -26.073,Z -220.849,A -90.000,B 90.000,C 0.000} C_DIS
LIN {X 86.848,Y -26.048,Z -223.337,A -90.000,B 90.000,C 0.000} C_DIS
LIN {X 86.425,Y -26.036,Z -225.092,A -90.000,B 90.000,C 0.000} C_DIS
LIN {X 86.312,Y -26.032,Z -225.541,A -90.000,B 90.000,C 0.000} C_DIS
LIN {X 85.727,Y -26.012,Z -227.822,A -90.000,B 90.000,C 0.000} C_DIS
LIN {X 84.945,Y -25.995,Z -230.899,A -90.000,B 90.000,C 0.000} C_DIS
LIN {X 84.878,Y -25.995,Z -231.145,A -90.000,B 90.000,C 0.000} C_DIS
LIN {X 84.799,Y -25.993,Z -231.419,A -90.000,B 90.000,C 0.000} C_DIS
LIN {X 84.196,Y -25.990,Z -233.472,A -90.000,B 90.000,C 0.000} C_DIS
LIN {X 83.203,Y -25.999,Z -236.898,A -90.000,B 90.000,C 0.000} C_DIS
LIN {X 83.159,Y -25.996,Z -237.040,A -90.000,B 90.000,C 0.000} C_DIS
LIN {X 82.577,Y -25.994,Z -238.762,A -90.000,B 90.000,C 0.000} C_DIS
LIN {X 81.186,Y -26.013,Z -242.928,A -90.000,B 90.000,C 0.000} C_DIS
LIN {X 81.126,Y -26.008,Z -243.097,A -90.000,B 90.000,C 0.000} C_DIS
LIN {X 81.095,Y -26.006,Z -243.180,A -90.000,B 90.000,C 0.000} C_DIS
LIN {X 80.945,Y -26.006,Z -243.561,A -90.000,B 90.000,C 0.000} C_DIS
LIN {X 80.945,Y -60.000,Z -243.561,A -90.000,B 90.000,C 0.000} C_DIS
LIN {X -104.795,Y -60.000,Z -243.561,A -90.000,B 90.000,C 0.000} C_DIS
LIN {X -104.795,Y -25.633,Z -243.561,A -90.000,B 90.000,C 0.000} C_DIS
LIN {X -104.580,Y -25.520,Z -243.386,A -90.000,B 90.000,C 0.000} C_DIS
LIN {X -104.091,Y -25.422,Z -243.022,A -90.000,B 90.000,C 0.000} C_DIS
LIN {X -102.165,Y -25.409,Z -241.680,A -90.000,B 90.000,C 0.000} C_DIS
LIN {X -101.815,Y -25.404,Z -241.448,A -90.000,B 90.000,C 0.000} C_DIS
LIN {X -101.290,Y -25.403,Z -241.101,A -90.000,B 90.000,C 0.000} C_DIS
LIN {X -99.060,Y -25.404,Z -239.602,A -90.000,B 90.000,C 0.000} C_DIS
LIN {X -94.267,Y -25.387,Z -236.376,A -90.000,B 90.000,C 0.000} C_DIS
LIN {X -94.091,Y -25.386,Z -236.262,A -90.000,B 90.000,C 0.000} C_DIS
LIN {X -91.828,Y -25.387,Z -234.793,A -90.000,B 90.000,C 0.000} C_DIS
LIN {X -86.127,Y -25.376,Z -231.089,A -90.000,B 90.000,C 0.000} C_DIS
LIN {X -85.503,Y -25.372,Z -230.699,A -90.000,B 90.000,C 0.000} C_DIS
LIN {X -83.295,Y -25.371,Z -229.319,A -90.000,B 90.000,C 0.000} C_DIS
LIN {X -81.347,Y -25.369,Z -228.106,A -90.000,B 90.000,C 0.000} C_DIS
LIN {X -77.837,Y -25.369,Z -225.922,A -90.000,B 90.000,C 0.000} C_DIS
LIN {X -77.273,Y -25.368,Z -225.572,A -90.000,B 90.000,C 0.000} C_DIS
LIN {X -70.404,Y -25.378,Z -221.474,A -90.000,B 90.000,C 0.000} C_DIS
LIN {X -68.665,Y -25.380,Z -220.440,A -90.000,B 90.000,C 0.000} C_DIS
LIN {X -63.103,Y -25.397,Z -217.220,A -90.000,B 90.000,C 0.000} C_DIS
LIN {X -62.499,Y -25.398,Z -216.873,A -90.000,B 90.000,C 0.000} C_DIS
LIN {X -60.438,Y -25.404,Z -215.689,A -90.000,B 90.000,C 0.000} C_DIS
LIN {X -57.046,Y -25.418,Z -213.763,A -90.000,B 90.000,C 0.000} C_DIS
LIN {X -53.948,Y -25.434,Z -212.006,A -90.000,B 90.000,C 0.000} C_DIS
LIN {X -52.541,Y -25.439,Z -211.223,A -90.000,B 90.000,C 0.000} C_DIS
LIN {X -47.807,Y -25.466,Z -208.558,A -90.000,B 90.000,C 0.000} C_DIS
LIN {X -46.982,Y -25.468,Z -208.102,A -90.000,B 90.000,C 0.000} C_DIS
LIN {X -45.416,Y -25.476,Z -207.240,A -90.000,B 90.000,C 0.000} C_DIS
LIN {X -41.620,Y -25.499,Z -205.083,A -90.000,B 90.000,C 0.000} C_DIS
LIN {X -40.275,Y -25.510,Z -204.322,A -90.000,B 90.000,C 0.000} C_DIS
LIN {X -39.802,Y -25.512,Z -204.059,A -90.000,B 90.000,C 0.000} C_DIS
LIN {X -39.563,Y -25.515,Z -203.921,A -90.000,B 90.000,C 0.000} C_DIS
LIN {X -36.358,Y -25.534,Z -202.053,A -90.000,B 90.000,C 0.000} C_DIS
LIN {X -35.118,Y -25.536,Z -201.342,A -90.000,B 90.000,C 0.000} C_DIS
LIN {X -34.804,Y -25.541,Z -201.152,A -90.000,B 90.000,C 0.000} C_DIS
LIN {X -32.840,Y -25.550,Z -199.947,A -90.000,B 90.000,C 0.000} C_DIS
LIN {X -31.076,Y -25.555,Z -198.872,A -90.000,B 90.000,C 0.000} C_DIS
LIN {X -30.793,Y -25.562,Z -198.690,A -90.000,B 90.000,C 0.000} C_DIS
LIN {X -29.270,Y -25.566,Z -197.682,A -90.000,B 90.000,C 0.000} C_DIS
LIN {X -27.758,Y -25.572,Z -196.682,A -90.000,B 90.000,C 0.000} C_DIS
LIN {X -27.657,Y -25.575,Z -196.611,A -90.000,B 90.000,C 0.000} C_DIS
LIN {X -25.053,Y -25.595,Z -194.727,A -90.000,B 90.000,C 0.000} C_DIS
LIN {X -24.514,Y -25.598,Z -194.335,A -90.000,B 90.000,C 0.000} C_DIS
LIN {X -24.400,Y -25.602,Z -194.247,A -90.000,B 90.000,C 0.000} C_DIS
LIN {X -23.307,Y -25.615,Z -193.376,A -90.000,B 90.000,C 0.000} C_DIS
LIN {X -21.742,Y -25.634,Z -192.104,A -90.000,B 90.000,C 0.000} C_DIS
LIN {X -21.662,Y -25.637,Z -192.036,A -90.000,B 90.000,C 0.000} C_DIS
LIN {X -20.660,Y -25.655,Z -191.163,A -90.000,B 90.000,C 0.000} C_DIS
LIN {X -18.993,Y -25.678,Z -189.675,A -90.000,B 90.000,C 0.000} C_DIS
LIN {X -18.712,Y -25.688,Z -189.413,A -90.000,B 90.000,C 0.000} C_DIS
LIN {X -18.530,Y -25.692,Z -189.242,A -90.000,B 90.000,C 0.000} C_DIS
LIN {X -17.066,Y -25.719,Z -187.821,A -90.000,B 90.000,C 0.000} C_DIS
LIN {X -16.310,Y -25.736,Z -187.083,A -90.000,B 90.000,C 0.000} C_DIS
LIN {X -16.128,Y -25.741,Z -186.896,A -90.000,B 90.000,C 0.000} C_DIS
LIN {X -14.867,Y -25.755,Z -185.572,A -90.000,B 90.000,C 0.000} C_DIS
LIN {X -14.538,Y -25.762,Z -185.231,A -90.000,B 90.000,C 0.000} C_DIS
LIN {X -13.972,Y -25.779,Z -184.637,A -90.000,B 90.000,C 0.000} C_DIS
LIN {X -13.500,Y -25.792,Z -184.142,A -90.000,B 90.000,C 0.000} C_DIS
LIN {X -13.141,Y -25.812,Z -183.752,A -90.000,B 90.000,C 0.000} C_DIS
LIN {X -12.289,Y -25.823,Z -182.781,A -90.000,B 90.000,C 0.000} C_DIS
LIN {X -11.792,Y -25.835,Z -182.204,A -90.000,B 90.000,C 0.000} C_DIS
LIN {X -10.942,Y -25.859,Z -181.220,A -90.000,B 90.000,C 0.000} C_DIS
LIN {X -10.545,Y -25.888,Z -180.736,A -90.000,B 90.000,C 0.000} C_DIS
LIN {X -8.942,Y -25.951,Z -178.675,A -90.000,B 90.000,C 0.000} C_DIS
LIN {X -8.563,Y -25.957,Z -178.171,A -90.000,B 90.000,C 0.000} C_DIS
LIN {X -8.437,Y -25.960,Z -178.002,A -90.000,B 90.000,C 0.000} C_DIS
LIN {X -8.018,Y -25.991,Z -177.405,A -90.000,B 90.000,C 0.000} C_DIS
LIN {X -7.852,Y -26.000,Z -177.161,A -90.000,B 90.000,C 0.000} C_DIS
LIN {X -7.485,Y -26.006,Z -176.592,A -90.000,B 90.000,C 0.000} C_DIS
LIN {X -7.038,Y -26.015,Z -175.906,A -90.000,B 90.000,C 0.000} C_DIS
LIN {X -6.291,Y -26.046,Z -174.737,A -90.000,B 90.000,C 0.000} C_DIS
LIN {X -6.115,Y -26.065,Z -174.445,A -90.000,B 90.000,C 0.000} C_DIS
LIN {X -6.067,Y -26.070,Z -174.364,A -90.000,B 90.000,C 0.000} C_DIS
LIN {X -5.639,Y -26.084,Z -173.567,A -90.000,B 90.000,C 0.000} C_DIS
LIN {X -4.970,Y -26.127,Z -172.289,A -90.000,B 90.000,C 0.000} C_DIS
LIN {X -4.541,Y -26.135,Z -171.407,A -90.000,B 90.000,C 0.000} C_DIS
LIN {X -4.367,Y -26.156,Z -171.022,A -90.000,B 90.000,C 0.000} C_DIS
LIN {X -4.335,Y -26.156,Z -170.934,A -90.000,B 90.000,C 0.000} C_DIS
LIN {X -4.152,Y -26.157,Z -170.392,A -90.000,B 90.000,C 0.000} C_DIS
LIN {X -3.340,Y -26.184,Z -168.084,A -90.000,B 90.000,C 0.000} C_DIS
LIN {X -3.289,Y -26.198,Z -167.913,A -90.000,B 90.000,C 0.000} C_DIS
LIN {X -3.006,Y -26.206,Z -166.406,A -90.000,B 90.000,C 0.000} C_DIS
LIN {X -2.814,Y -26.193,Z -165.250,A -90.000,B 90.000,C 0.000} C_DIS
LIN {X -2.814,Y -26.190,Z -165.223,A -90.000,B 90.000,C 0.000} C_DIS
LIN {X -2.826,Y -26.188,Z -165.009,A -90.000,B 90.000,C 0.000} C_DIS
LIN {X -2.901,Y -26.168,Z -163.839,A -90.000,B 90.000,C 0.000} C_DIS
LIN {X -2.930,Y -26.156,Z -163.353,A -90.000,B 90.000,C 0.000} C_DIS
LIN {X -3.052,Y -26.074,Z -162.911,A -90.000,B 90.000,C 0.000} C_DIS
LIN {X -3.122,Y -26.069,Z -162.737,A -90.000,B 90.000,C 0.000} C_DIS
LIN {X -3.172,Y -26.068,Z -162.605,A -90.000,B 90.000,C 0.000} C_DIS
LIN {X -3.396,Y -26.057,Z -161.993,A -90.000,B 90.000,C 0.000} C_DIS
LIN {X -3.568,Y -26.003,Z -161.694,A -90.000,B 90.000,C 0.000} C_DIS
LIN {X -3.766,Y -25.941,Z -161.342,A -90.000,B 90.000,C 0.000} C_DIS
LIN {X -3.783,Y -25.941,Z -161.319,A -90.000,B 90.000,C 0.000} C_DIS
LIN {X -4.136,Y -25.924,Z -160.823,A -90.000,B 90.000,C 0.000} C_DIS
LIN {X -4.259,Y -25.898,Z -160.684,A -90.000,B 90.000,C 0.000} C_DIS
LIN {X -4.673,Y -25.815,Z -160.210,A -90.000,B 90.000,C 0.000} C_DIS
LIN {X -4.777,Y -25.795,Z -160.082,A -90.000,B 90.000,C 0.000} C_DIS
LIN {X -5.308,Y -25.791,Z -159.575,A -90.000,B 90.000,C 0.000} C_DIS
LIN {X -5.645,Y -25.753,Z -159.295,A -90.000,B 90.000,C 0.000} C_DIS
LIN {X -5.922,Y -25.714,Z -159.050,A -90.000,B 90.000,C 0.000} C_DIS
LIN {X -6.025,Y -25.702,Z -158.956,A -90.000,B 90.000,C 0.000} C_DIS
LIN {X -6.594,Y -25.702,Z -158.532,A -90.000,B 90.000,C 0.000} C_DIS
LIN {X -7.082,Y -25.688,Z -158.145,A -90.000,B 90.000,C 0.000} C_DIS
LIN {X -7.593,Y -25.656,Z -157.755,A -90.000,B 90.000,C 0.000} C_DIS
LIN {X -8.030,Y -25.643,Z -157.443,A -90.000,B 90.000,C 0.000} C_DIS
LIN {X -8.769,Y -25.631,Z -156.907,A -90.000,B 90.000,C 0.000} C_DIS
LIN {X -9.531,Y -25.608,Z -156.344,A -90.000,B 90.000,C 0.000} C_DIS
LIN {X -10.166,Y -25.596,Z -155.888,A -90.000,B 90.000,C 0.000} C_DIS
LIN {X -11.467,Y -25.562,Z -154.929,A -90.000,B 90.000,C 0.000} C_DIS
LIN {X -11.606,Y -25.561,Z -154.824,A -90.000,B 90.000,C 0.000} C_DIS
LIN {X -12.055,Y -25.552,Z -154.466,A -90.000,B 90.000,C 0.000} C_DIS
LIN {X -13.873,Y -25.517,Z -153.100,A -90.000,B 90.000,C 0.000} C_DIS
LIN {X -13.939,Y -25.515,Z -153.047,A -90.000,B 90.000,C 0.000} C_DIS
LIN {X -14.378,Y -25.510,Z -152.688,A -90.000,B 90.000,C 0.000} C_DIS
LIN {X -16.492,Y -25.483,Z -151.036,A -90.000,B 90.000,C 0.000} C_DIS
LIN {X -16.631,Y -25.479,Z -150.921,A -90.000,B 90.000,C 0.000} C_DIS
LIN {X -17.066,Y -25.477,Z -150.556,A -90.000,B 90.000,C 0.000} C_DIS
LIN {X -18.950,Y -25.465,Z -149.005,A -90.000,B 90.000,C 0.000} C_DIS
LIN {X -19.532,Y -25.455,Z -148.529,A -90.000,B 90.000,C 0.000} C_DIS
LIN {X -19.891,Y -25.449,Z -148.231,A -90.000,B 90.000,C 0.000} C_DIS
LIN {X -20.050,Y -25.444,Z -148.090,A -90.000,B 90.000,C 0.000} C_DIS
LIN {X -21.355,Y -25.430,Z -146.918,A -90.000,B 90.000,C 0.000} C_DIS
LIN {X -22.195,Y -25.417,Z -146.167,A -90.000,B 90.000,C 0.000} C_DIS
LIN {X -23.129,Y -25.404,Z -145.338,A -90.000,B 90.000,C 0.000} C_DIS
LIN {X -23.372,Y -25.393,Z -145.100,A -90.000,B 90.000,C 0.000} C_DIS
LIN {X -25.945,Y -25.346,Z -142.516,A -90.000,B 90.000,C 0.000} C_DIS
LIN {X -26.675,Y -25.331,Z -141.782,A -90.000,B 90.000,C 0.000} C_DIS
LIN {X -27.120,Y -25.320,Z -141.250,A -90.000,B 90.000,C 0.000} C_DIS
LIN {X -27.590,Y -25.314,Z -140.687,A -90.000,B 90.000,C 0.000} C_DIS
LIN {X -28.721,Y -25.309,Z -139.405,A -90.000,B 90.000,C 0.000} C_DIS
LIN {X -29.254,Y -25.308,Z -138.812,A -90.000,B 90.000,C 0.000} C_DIS
LIN {X -29.371,Y -25.308,Z -138.703,A -90.000,B 90.000,C 0.000} C_DIS
LIN {X -29.419,Y -25.308,Z -138.650,A -90.000,B 90.000,C 0.000} C_DIS
LIN {X -29.421,Y -28.521,Z -138.648,A -90.000,B 90.000,C 0.000} C_DIS
LIN {X -29.422,Y -28.546,Z -138.647,A -90.000,B 90.000,C 0.000} C_DIS
LIN {X -29.431,Y -28.594,Z -138.637,A -90.000,B 90.000,C 0.000} C_DIS
LIN {X -29.442,Y -28.628,Z -138.625,A -90.000,B 90.000,C 0.000} C_DIS
LIN {X -29.464,Y -28.671,Z -138.600,A -90.000,B 90.000,C 0.000} C_DIS
LIN {X -29.546,Y -28.756,Z -138.512,A -90.000,B 90.000,C 0.000} C_DIS
LIN {X -29.617,Y -28.793,Z -138.436,A -90.000,B 90.000,C 0.000} C_DIS
LIN {X -29.728,Y -28.808,Z -138.320,A -90.000,B 90.000,C 0.000} C_DIS
LIN {X -29.770,Y -28.796,Z -138.278,A -90.000,B 90.000,C 0.000} C_DIS
LIN {X -29.805,Y -28.775,Z -138.245,A -90.000,B 90.000,C 0.000} C_DIS
LIN {X -29.830,Y -28.748,Z -138.221,A -90.000,B 90.000,C 0.000} C_DIS
LIN {X -29.850,Y -28.717,Z -138.204,A -90.000,B 90.000,C 0.000} C_DIS
LIN {X -29.864,Y -28.682,Z -138.192,A -90.000,B 90.000,C 0.000} C_DIS
LIN {X -29.874,Y -28.643,Z -138.185,A -90.000,B 90.000,C 0.000} C_DIS
LIN {X -29.880,Y -28.600,Z -138.182,A -90.000,B 90.000,C 0.000} C_DIS
LIN {X -29.883,Y -28.550,Z -138.181,A -90.000,B 90.000,C 0.000} C_DIS
LIN {X -29.886,Y -25.306,Z -138.182,A -90.000,B 90.000,C 0.000} C_DIS
LIN {X -29.898,Y -25.308,Z -138.175,A -90.000,B 90.000,C 0.000} C_DIS
LIN {X -29.907,Y -25.308,Z -138.175,A -90.000,B 90.000,C 0.000} C_DIS
LIN {X -29.926,Y -25.308,Z -138.163,A -90.000,B 90.000,C 0.000} C_DIS
LIN {X -29.987,Y -25.308,Z -138.103,A -90.000,B 90.000,C 0.000} C_DIS
LIN {X -30.165,Y -25.308,Z -137.903,A -90.000,B 90.000,C 0.000} C_DIS
LIN {X -30.320,Y -25.307,Z -137.740,A -90.000,B 90.000,C 0.000} C_DIS
LIN {X -30.505,Y -25.308,Z -137.505,A -90.000,B 90.000,C 0.000} C_DIS
LIN {X -30.527,Y -25.308,Z -137.478,A -90.000,B 90.000,C 0.000} C_DIS
LIN {X -30.801,Y -25.308,Z -137.155,A -90.000,B 90.000,C 0.000} C_DIS
LIN {X -31.254,Y -25.308,Z -136.631,A -90.000,B 90.000,C 0.000} C_DIS
LIN {X -31.437,Y -25.308,Z -136.424,A -90.000,B 90.000,C 0.000} C_DIS
LIN {X -31.726,Y -25.308,Z -136.106,A -90.000,B 90.000,C 0.000} C_DIS
LIN {X -31.926,Y -25.308,Z -135.899,A -90.000,B 90.000,C 0.000} C_DIS
LIN {X -32.055,Y -25.308,Z -135.778,A -90.000,B 90.000,C 0.000} C_DIS
LIN {X -32.098,Y -25.308,Z -135.743,A -90.000,B 90.000,C 0.000} C_DIS
LIN {X -32.141,Y -25.308,Z -135.715,A -90.000,B 90.000,C 0.000} C_DIS
LIN {X -32.165,Y -25.308,Z -135.707,A -90.000,B 90.000,C 0.000} C_DIS
LIN {X -32.187,Y -25.308,Z -135.715,A -90.000,B 90.000,C 0.000} C_DIS
LIN {X -32.199,Y -25.308,Z -135.705,A -90.000,B 90.000,C 0.000} C_DIS
LIN {X -32.264,Y -25.308,Z -135.615,A -90.000,B 90.000,C 0.000} C_DIS
LIN {X -32.758,Y -25.308,Z -134.874,A -90.000,B 90.000,C 0.000} C_DIS
LIN {X -33.539,Y -25.308,Z -133.722,A -90.000,B 90.000,C 0.000} C_DIS
LIN {X -33.583,Y -25.308,Z -133.658,A -90.000,B 90.000,C 0.000} C_DIS
LIN {X -33.873,Y -25.308,Z -133.234,A -90.000,B 90.000,C 0.000} C_DIS
LIN {X -34.353,Y -25.306,Z -132.544,A -90.000,B 90.000,C 0.000} C_DIS
LIN {X -34.546,Y -25.305,Z -132.271,A -90.000,B 90.000,C 0.000} C_DIS
LIN {X -34.852,Y -25.301,Z -131.850,A -90.000,B 90.000,C 0.000} C_DIS
LIN {X -35.064,Y -25.296,Z -131.572,A -90.000,B 90.000,C 0.000} C_DIS
LIN {X -35.199,Y -25.291,Z -131.408,A -90.000,B 90.000,C 0.000} C_DIS
LIN {X -35.244,Y -25.288,Z -131.359,A -90.000,B 90.000,C 0.000} C_DIS
LIN {X -35.298,Y -25.283,Z -131.310,A -90.000,B 90.000,C 0.000} C_DIS
LIN {X -35.312,Y -25.280,Z -131.302,A -90.000,B 90.000,C 0.000} C_DIS
LIN {X -35.328,Y -25.274,Z -131.303,A -90.000,B 90.000,C 0.000} C_DIS
LIN {X -35.332,Y -25.273,Z -131.299,A -90.000,B 90.000,C 0.000} C_DIS
LIN {X -35.400,Y -25.270,Z -131.166,A -90.000,B 90.000,C 0.000} C_DIS
LIN {X -35.495,Y -25.272,Z -130.977,A -90.000,B 90.000,C 0.000} C_DIS
LIN {X -35.899,Y -25.284,Z -130.208,A -90.000,B 90.000,C 0.000} C_DIS
LIN {X -36.063,Y -25.288,Z -129.916,A -90.000,B 90.000,C 0.000} C_DIS
LIN {X -36.463,Y -25.300,Z -129.178,A -90.000,B 90.000,C 0.000} C_DIS
LIN {X -36.704,Y -25.308,Z -128.724,A -90.000,B 90.000,C 0.000} C_DIS
LIN {X -37.294,Y -25.327,Z -127.647,A -90.000,B 90.000,C 0.000} C_DIS
LIN {X -37.314,Y -25.333,Z -127.610,A -90.000,B 90.000,C 0.000} C_DIS
LIN {X -37.546,Y -25.332,Z -127.187,A -90.000,B 90.000,C 0.000} C_DIS
LIN {X -38.004,Y -25.308,Z -126.352,A -90.000,B 90.000,C 0.000} C_DIS
LIN {X -38.234,Y -25.309,Z -125.927,A -90.000,B 90.000,C 0.000} C_DIS
LIN {X -38.970,Y -25.309,Z -124.276,A -90.000,B 90.000,C 0.000} C_DIS
LIN {X -39.697,Y -25.311,Z -122.799,A -90.000,B 90.000,C 0.000} C_DIS
LIN {X -39.732,Y -25.311,Z -122.727,A -90.000,B 90.000,C 0.000} C_DIS
LIN {X -40.349,Y -25.314,Z -121.319,A -90.000,B 90.000,C 0.000} C_DIS
LIN {X -40.676,Y -25.320,Z -120.569,A -90.000,B 90.000,C 0.000} C_DIS
LIN {X -40.863,Y -25.327,Z -120.128,A -90.000,B 90.000,C 0.000} C_DIS
LIN {X -41.120,Y -25.332,Z -119.369,A -90.000,B 90.000,C 0.000} C_DIS
LIN {X -41.565,Y -25.355,Z -118.259,A -90.000,B 90.000,C 0.000} C_DIS
LIN {X -41.684,Y -25.363,Z -117.960,A -90.000,B 90.000,C 0.000} C_DIS
LIN {X -41.912,Y -25.372,Z -117.299,A -90.000,B 90.000,C 0.000} C_DIS
LIN {X -42.392,Y -25.417,Z -116.229,A -90.000,B 90.000,C 0.000} C_DIS
LIN {X -42.444,Y -25.423,Z -116.111,A -90.000,B 90.000,C 0.000} C_DIS
LIN {X -42.538,Y -25.431,Z -115.883,A -90.000,B 90.000,C 0.000} C_DIS
LIN {X -42.593,Y -25.435,Z -115.747,A -90.000,B 90.000,C 0.000} C_DIS
LIN {X -42.672,Y -25.438,Z -115.558,A -90.000,B 90.000,C 0.000} C_DIS
LIN {X -43.352,Y -25.513,Z -114.280,A -90.000,B 90.000,C 0.000} C_DIS
LIN {X -43.712,Y -25.522,Z -113.606,A -90.000,B 90.000,C 0.000} C_DIS
LIN {X -43.922,Y -25.540,Z -113.270,A -90.000,B 90.000,C 0.000} C_DIS
LIN {X -44.442,Y -25.578,Z -112.447,A -90.000,B 90.000,C 0.000} C_DIS
LIN {X -44.970,Y -25.587,Z -111.642,A -90.000,B 90.000,C 0.000} C_DIS
LIN {X -45.272,Y -25.585,Z -111.188,A -90.000,B 90.000,C 0.000} C_DIS
LIN {X -45.964,Y -25.602,Z -110.210,A -90.000,B 90.000,C 0.000} C_DIS
LIN {X -46.169,Y -25.605,Z -109.928,A -90.000,B 90.000,C 0.000} C_DIS
LIN {X -47.412,Y -25.598,Z -108.244,A -90.000,B 90.000,C 0.000} C_DIS
LIN {X -47.489,Y -25.597,Z -108.139,A -90.000,B 90.000,C 0.000} C_DIS
LIN {X -47.921,Y -25.599,Z -107.560,A -90.000,B 90.000,C 0.000} C_DIS
LIN {X -48.904,Y -25.594,Z -106.252,A -90.000,B 90.000,C 0.000} C_DIS
LIN {X -49.418,Y -25.602,Z -105.597,A -90.000,B 90.000,C 0.000} C_DIS
LIN {X -49.599,Y -25.601,Z -105.369,A -90.000,B 90.000,C 0.000} C_DIS
LIN {X -50.006,Y -25.590,Z -104.843,A -90.000,B 90.000,C 0.000} C_DIS
LIN {X -50.605,Y -25.588,Z -104.058,A -90.000,B 90.000,C 0.000} C_DIS
LIN {X -50.742,Y -25.590,Z -103.884,A -90.000,B 90.000,C 0.000} C_DIS
LIN {X -52.110,Y -25.583,Z -102.179,A -90.000,B 90.000,C 0.000} C_DIS
LIN {X -52.521,Y -25.576,Z -101.649,A -90.000,B 90.000,C 0.000} C_DIS
LIN {X -53.044,Y -25.578,Z -100.965,A -90.000,B 90.000,C 0.000} C_DIS
LIN {X -53.335,Y -25.577,Z -100.579,A -90.000,B 90.000,C 0.000} C_DIS
LIN {X -53.985,Y -25.572,Z -99.710,A -90.000,B 90.000,C 0.000} C_DIS
LIN {X -54.129,Y -25.573,Z -99.516,A -90.000,B 90.000,C 0.000} C_DIS
LIN {X -54.473,Y -25.579,Z -99.068,A -90.000,B 90.000,C 0.000} C_DIS
LIN {X -54.541,Y -25.580,Z -98.977,A -90.000,B 90.000,C 0.000} C_DIS
LIN {X -54.747,Y -25.581,Z -98.703,A -90.000,B 90.000,C 0.000} C_DIS
LIN {X -55.036,Y -25.577,Z -98.314,A -90.000,B 90.000,C 0.000} C_DIS
LIN {X -55.866,Y -25.581,Z -97.181,A -90.000,B 90.000,C 0.000} C_DIS
LIN {X -56.354,Y -25.591,Z -96.536,A -90.000,B 90.000,C 0.000} C_DIS
LIN {X -56.912,Y -25.593,Z -95.801,A -90.000,B 90.000,C 0.000} C_DIS
LIN {X -57.197,Y -25.592,Z -95.420,A -90.000,B 90.000,C 0.000} C_DIS
LIN {X -57.833,Y -25.600,Z -94.581,A -90.000,B 90.000,C 0.000} C_DIS
LIN {X -58.777,Y -25.605,Z -93.337,A -90.000,B 90.000,C 0.000} C_DIS
LIN {X -59.019,Y -25.605,Z -93.016,A -90.000,B 90.000,C 0.000} C_DIS
LIN {X -59.271,Y -25.603,Z -92.674,A -90.000,B 90.000,C 0.000} C_DIS
LIN {X -59.656,Y -25.602,Z -92.163,A -90.000,B 90.000,C 0.000} C_DIS
LIN {X -60.454,Y -25.608,Z -91.093,A -90.000,B 90.000,C 0.000} C_DIS
LIN {X -61.084,Y -25.623,Z -90.276,A -90.000,B 90.000,C 0.000} C_DIS
LIN {X -61.403,Y -25.638,Z -89.879,A -90.000,B 90.000,C 0.000} C_DIS
LIN {X -62.279,Y -25.646,Z -88.820,A -90.000,B 90.000,C 0.000} C_DIS
LIN {X -62.525,Y -25.646,Z -88.516,A -90.000,B 90.000,C 0.000} C_DIS
LIN {X -62.996,Y -25.650,Z -87.932,A -90.000,B 90.000,C 0.000} C_DIS
LIN {X -63.234,Y -25.660,Z -87.655,A -90.000,B 90.000,C 0.000} C_DIS
LIN {X -64.612,Y -25.665,Z -86.097,A -90.000,B 90.000,C 0.000} C_DIS
LIN {X -64.834,Y -25.664,Z -85.842,A -90.000,B 90.000,C 0.000} C_DIS
LIN {X -65.037,Y -25.667,Z -85.613,A -90.000,B 90.000,C 0.000} C_DIS
LIN {X -66.164,Y -25.664,Z -84.359,A -90.000,B 90.000,C 0.000} C_DIS
LIN {X -66.530,Y -25.671,Z -83.945,A -90.000,B 90.000,C 0.000} C_DIS
LIN {X -67.763,Y -25.713,Z -82.581,A -90.000,B 90.000,C 0.000} C_DIS
LIN {X -68.052,Y -25.724,Z -82.256,A -90.000,B 90.000,C 0.000} C_DIS
LIN {X -68.477,Y -25.725,Z -81.793,A -90.000,B 90.000,C 0.000} C_DIS
LIN {X -69.149,Y -25.743,Z -81.061,A -90.000,B 90.000,C 0.000} C_DIS
LIN {X -70.047,Y -25.765,Z -80.070,A -90.000,B 90.000,C 0.000} C_DIS
LIN {X -70.347,Y -25.773,Z -79.738,A -90.000,B 90.000,C 0.000} C_DIS
LIN {X -70.823,Y -25.778,Z -79.191,A -90.000,B 90.000,C 0.000} C_DIS
LIN {X -71.666,Y -25.805,Z -78.201,A -90.000,B 90.000,C 0.000} C_DIS
LIN {X -71.955,Y -25.822,Z -77.875,A -90.000,B 90.000,C 0.000} C_DIS
LIN {X -73.006,Y -25.849,Z -76.738,A -90.000,B 90.000,C 0.000} C_DIS
LIN {X -73.457,Y -25.878,Z -76.259,A -90.000,B 90.000,C 0.000} C_DIS
LIN {X -74.075,Y -25.900,Z -75.626,A -90.000,B 90.000,C 0.000} C_DIS
LIN {X -74.481,Y -25.933,Z -75.236,A -90.000,B 90.000,C 0.000} C_DIS
LIN {X -74.790,Y -25.940,Z -74.964,A -90.000,B 90.000,C 0.000} C_DIS
LIN {X -74.940,Y -25.958,Z -74.850,A -90.000,B 90.000,C 0.000} C_DIS
LIN {X -75.028,Y -25.982,Z -74.802,A -90.000,B 90.000,C 0.000} C_DIS
LIN {X -75.066,Y -25.996,Z -74.786,A -90.000,B 90.000,C 0.000} C_DIS
LIN {X -75.152,Y -26.033,Z -74.752,A -90.000,B 90.000,C 0.000} C_DIS
LIN {X -75.207,Y -26.052,Z -74.726,A -90.000,B 90.000,C 0.000} C_DIS
LIN {X -75.340,Y -26.091,Z -74.673,A -90.000,B 90.000,C 0.000} C_DIS
LIN {X -75.479,Y -26.089,Z -74.666,A -90.000,B 90.000,C 0.000} C_DIS
LIN {X -75.705,Y -26.095,Z -74.662,A -90.000,B 90.000,C 0.000} C_DIS
LIN {X -75.898,Y -26.096,Z -74.662,A -90.000,B 90.000,C 0.000} C_DIS
LIN {X -76.284,Y -26.086,Z -74.649,A -90.000,B 90.000,C 0.000} C_DIS
LIN {X -76.361,Y -26.083,Z -74.645,A -90.000,B 90.000,C 0.000} C_DIS
LIN {X -76.505,Y -26.080,Z -74.639,A -90.000,B 90.000,C 0.000} C_DIS
LIN {X -76.744,Y -26.066,Z -74.619,A -90.000,B 90.000,C 0.000} C_DIS
LIN {X -76.997,Y -26.054,Z -74.594,A -90.000,B 90.000,C 0.000} C_DIS
LIN {X -77.515,Y -26.048,Z -74.547,A -90.000,B 90.000,C 0.000} C_DIS
LIN {X -77.828,Y -26.032,Z -74.505,A -90.000,B 90.000,C 0.000} C_DIS
LIN {X -77.993,Y -26.027,Z -74.479,A -90.000,B 90.000,C 0.000} C_DIS
LIN {X -78.471,Y -25.990,Z -74.369,A -90.000,B 90.000,C 0.000} C_DIS
LIN {X -78.674,Y -25.980,Z -74.316,A -90.000,B 90.000,C 0.000} C_DIS
LIN {X -79.055,Y -25.966,Z -74.210,A -90.000,B 90.000,C 0.000} C_DIS
LIN {X -79.417,Y -25.959,Z -74.100,A -90.000,B 90.000,C 0.000} C_DIS
LIN {X -79.615,Y -25.956,Z -74.037,A -90.000,B 90.000,C 0.000} C_DIS
LIN {X -80.148,Y -25.925,Z -73.835,A -90.000,B 90.000,C 0.000} C_DIS
LIN {X -80.414,Y -25.914,Z -73.730,A -90.000,B 90.000,C 0.000} C_DIS
LIN {X -80.544,Y -25.903,Z -73.671,A -90.000,B 90.000,C 0.000} C_DIS
LIN {X -80.741,Y -25.892,Z -73.570,A -90.000,B 90.000,C 0.000} C_DIS
LIN {X -81.024,Y -25.876,Z -73.422,A -90.000,B 90.000,C 0.000} C_DIS
LIN {X -81.130,Y -25.872,Z -73.365,A -90.000,B 90.000,C 0.000} C_DIS
LIN {X -81.305,Y -25.859,Z -73.263,A -90.000,B 90.000,C 0.000} C_DIS
LIN {X -81.426,Y -25.853,Z -73.189,A -90.000,B 90.000,C 0.000} C_DIS
LIN {X -81.878,Y -25.844,Z -72.901,A -90.000,B 90.000,C 0.000} C_DIS
LIN {X -81.979,Y -25.842,Z -72.835,A -90.000,B 90.000,C 0.000} C_DIS
LIN {X -82.041,Y -25.839,Z -72.793,A -90.000,B 90.000,C 0.000} C_DIS
LIN {X -82.177,Y -25.837,Z -72.694,A -90.000,B 90.000,C 0.000} C_DIS
LIN {X -82.320,Y -25.841,Z -72.583,A -90.000,B 90.000,C 0.000} C_DIS
LIN {X -82.537,Y -25.832,Z -72.393,A -90.000,B 90.000,C 0.000} C_DIS
LIN {X -82.744,Y -25.830,Z -72.205,A -90.000,B 90.000,C 0.000} C_DIS
LIN {X -82.934,Y -25.823,Z -72.036,A -90.000,B 90.000,C 0.000} C_DIS
LIN {X -83.023,Y -25.817,Z -71.951,A -90.000,B 90.000,C 0.000} C_DIS
LIN {X -83.114,Y -25.814,Z -71.861,A -90.000,B 90.000,C 0.000} C_DIS
LIN {X -83.212,Y -25.815,Z -71.759,A -90.000,B 90.000,C 0.000} C_DIS
LIN {X -83.382,Y -25.801,Z -71.560,A -90.000,B 90.000,C 0.000} C_DIS
LIN {X -83.492,Y -25.797,Z -71.422,A -90.000,B 90.000,C 0.000} C_DIS
LIN {X -83.844,Y -25.796,Z -70.946,A -90.000,B 90.000,C 0.000} C_DIS
LIN {X -83.939,Y -25.795,Z -70.818,A -90.000,B 90.000,C 0.000} C_DIS
LIN {X -84.087,Y -25.785,Z -70.587,A -90.000,B 90.000,C 0.000} C_DIS
LIN {X -84.153,Y -25.783,Z -70.481,A -90.000,B 90.000,C 0.000} C_DIS
LIN {X -84.177,Y -25.784,Z -70.439,A -90.000,B 90.000,C 0.000} C_DIS
LIN {X -84.377,Y -25.770,Z -70.053,A -90.000,B 90.000,C 0.000} C_DIS
LIN {X -84.473,Y -25.780,Z -69.857,A -90.000,B 90.000,C 0.000} C_DIS
LIN {X -84.535,Y -25.783,Z -69.716,A -90.000,B 90.000,C 0.000} C_DIS
LIN {X -84.659,Y -25.779,Z -69.451,A -90.000,B 90.000,C 0.000} C_DIS
LIN {X -84.706,Y -25.773,Z -69.328,A -90.000,B 90.000,C 0.000} C_DIS
LIN {X -84.830,Y -25.768,Z -68.960,A -90.000,B 90.000,C 0.000} C_DIS
LIN {X -84.879,Y -25.767,Z -68.805,A -90.000,B 90.000,C 0.000} C_DIS
LIN {X -84.911,Y -25.770,Z -68.694,A -90.000,B 90.000,C 0.000} C_DIS
LIN {X -84.971,Y -25.780,Z -68.488,A -90.000,B 90.000,C 0.000} C_DIS
LIN {X -85.004,Y -25.774,Z -68.354,A -90.000,B 90.000,C 0.000} C_DIS
LIN {X -85.054,Y -25.771,Z -68.132,A -90.000,B 90.000,C 0.000} C_DIS
LIN {X -85.093,Y -25.770,Z -67.953,A -90.000,B 90.000,C 0.000} C_DIS
LIN {X -85.119,Y -25.763,Z -67.801,A -90.000,B 90.000,C 0.000} C_DIS
LIN {X -85.135,Y -25.763,Z -67.688,A -90.000,B 90.000,C 0.000} C_DIS
LIN {X -85.150,Y -25.765,Z -67.574,A -90.000,B 90.000,C 0.000} C_DIS
LIN {X -85.179,Y -25.755,Z -67.435,A -90.000,B 90.000,C 0.000} C_DIS
LIN {X -85.225,Y -25.732,Z -67.173,A -90.000,B 90.000,C 0.000} C_DIS
LIN {X -85.251,Y -25.723,Z -67.001,A -90.000,B 90.000,C 0.000} C_DIS
LIN {X -85.271,Y -25.695,Z -66.727,A -90.000,B 90.000,C 0.000} C_DIS
LIN {X -85.291,Y -25.679,Z -66.528,A -90.000,B 90.000,C 0.000} C_DIS
LIN {X -85.346,Y -25.692,Z -66.326,A -90.000,B 90.000,C 0.000} C_DIS
LIN {X -85.371,Y -25.699,Z -66.230,A -90.000,B 90.000,C 0.000} C_DIS
LIN {X -85.438,Y -25.724,Z -66.009,A -90.000,B 90.000,C 0.000} C_DIS
LIN {X -85.637,Y -25.804,Z -65.447,A -90.000,B 90.000,C 0.000} C_DIS
LIN {X -85.667,Y -25.813,Z -65.377,A -90.000,B 90.000,C 0.000} C_DIS
LIN {X -85.695,Y -25.819,Z -65.317,A -90.000,B 90.000,C 0.000} C_DIS
LIN {X -85.925,Y -25.896,Z -64.888,A -90.000,B 90.000,C 0.000} C_DIS
LIN {X -85.946,Y -25.904,Z -64.847,A -90.000,B 90.000,C 0.000} C_DIS
LIN {X -86.049,Y -25.947,Z -64.656,A -90.000,B 90.000,C 0.000} C_DIS
LIN {X -86.127,Y -25.978,Z -64.502,A -90.000,B 90.000,C 0.000} C_DIS
LIN {X -86.172,Y -26.000,Z -64.409,A -90.000,B 90.000,C 0.000} C_DIS
LIN {X -86.366,Y -26.097,Z -63.978,A -90.000,B 90.000,C 0.000} C_DIS
LIN {X -86.447,Y -26.142,Z -63.799,A -90.000,B 90.000,C 0.000} C_DIS
LIN {X -86.468,Y -26.154,Z -63.752,A -90.000,B 90.000,C 0.000} C_DIS
LIN {X -86.519,Y -26.174,Z -63.663,A -90.000,B 90.000,C 0.000} C_DIS
LIN {X -86.625,Y -26.192,Z -63.555,A -90.000,B 90.000,C 0.000} C_DIS
LIN {X -86.887,Y -26.231,Z -63.272,A -90.000,B 90.000,C 0.000} C_DIS
LIN {X -87.533,Y -26.291,Z -62.672,A -90.000,B 90.000,C 0.000} C_DIS
LIN {X -87.590,Y -26.294,Z -62.618,A -90.000,B 90.000,C 0.000} C_DIS
LIN {X -88.204,Y -26.311,Z -62.058,A -90.000,B 90.000,C 0.000} C_DIS
LIN {X -88.603,Y -26.316,Z -61.689,A -90.000,B 90.000,C 0.000} C_DIS
LIN {X -88.827,Y -26.316,Z -61.480,A -90.000,B 90.000,C 0.000} C_DIS
LIN {X -89.074,Y -26.314,Z -61.256,A -90.000,B 90.000,C 0.000} C_DIS
LIN {X -89.821,Y -26.291,Z -60.566,A -90.000,B 90.000,C 0.000} C_DIS
LIN {X -90.230,Y -26.277,Z -60.182,A -90.000,B 90.000,C 0.000} C_DIS
LIN {X -90.414,Y -26.271,Z -60.003,A -90.000,B 90.000,C 0.000} C_DIS
LIN {X -90.591,Y -26.263,Z -59.828,A -90.000,B 90.000,C 0.000} C_DIS
LIN {X -91.041,Y -26.244,Z -59.375,A -90.000,B 90.000,C 0.000} C_DIS
LIN {X -91.732,Y -26.198,Z -58.664,A -90.000,B 90.000,C 0.000} C_DIS
LIN {X -91.879,Y -26.187,Z -58.509,A -90.000,B 90.000,C 0.000} C_DIS
LIN {X -92.100,Y -26.171,Z -58.272,A -90.000,B 90.000,C 0.000} C_DIS
LIN {X -92.310,Y -26.156,Z -58.041,A -90.000,B 90.000,C 0.000} C_DIS
LIN {X -92.488,Y -26.140,Z -57.842,A -90.000,B 90.000,C 0.000} C_DIS
LIN {X -92.943,Y -26.094,Z -57.297,A -90.000,B 90.000,C 0.000} C_DIS
LIN {X -93.370,Y -26.033,Z -56.729,A -90.000,B 90.000,C 0.000} C_DIS
LIN {X -93.478,Y -26.013,Z -56.580,A -90.000,B 90.000,C 0.000} C_DIS
LIN {X -93.500,Y -26.010,Z -56.549,A -90.000,B 90.000,C 0.000} C_DIS
LIN {X -93.850,Y -26.040,Z -56.180,A -90.000,B 90.000,C 0.000} C_DIS
LIN {X -94.021,Y -26.064,Z -55.986,A -90.000,B 90.000,C 0.000} C_DIS
LIN {X -94.108,Y -26.072,Z -55.884,A -90.000,B 90.000,C 0.000} C_DIS
LIN {X -94.432,Y -26.106,Z -55.501,A -90.000,B 90.000,C 0.000} C_DIS
LIN {X -94.793,Y -26.150,Z -55.064,A -90.000,B 90.000,C 0.000} C_DIS
LIN {X -94.830,Y -26.153,Z -55.015,A -90.000,B 90.000,C 0.000} C_DIS
LIN {X -94.933,Y -26.165,Z -54.874,A -90.000,B 90.000,C 0.000} C_DIS
LIN {X -95.358,Y -26.239,Z -54.245,A -90.000,B 90.000,C 0.000} C_DIS
LIN {X -95.498,Y -26.271,Z -54.018,A -90.000,B 90.000,C 0.000} C_DIS
LIN {X -95.601,Y -26.296,Z -53.845,A -90.000,B 90.000,C 0.000} C_DIS
LIN {X -95.701,Y -26.313,Z -53.666,A -90.000,B 90.000,C 0.000} C_DIS
LIN {X -95.738,Y -26.321,Z -53.597,A -90.000,B 90.000,C 0.000} C_DIS
LIN {X -95.892,Y -26.366,Z -53.277,A -90.000,B 90.000,C 0.000} C_DIS
LIN {X -96.018,Y -26.404,Z -53.008,A -90.000,B 90.000,C 0.000} C_DIS
LIN {X -96.065,Y -26.416,Z -52.904,A -90.000,B 90.000,C 0.000} C_DIS
LIN {X -96.126,Y -26.435,Z -52.755,A -90.000,B 90.000,C 0.000} C_DIS
LIN {X -96.191,Y -26.457,Z -52.587,A -90.000,B 90.000,C 0.000} C_DIS
LIN {X -96.295,Y -26.482,Z -52.298,A -90.000,B 90.000,C 0.000} C_DIS
LIN {X -96.365,Y -26.493,Z -52.092,A -90.000,B 90.000,C 0.000} C_DIS
LIN {X -96.397,Y -26.500,Z -51.992,A -90.000,B 90.000,C 0.000} C_DIS
LIN {X -96.423,Y -26.509,Z -51.897,A -90.000,B 90.000,C 0.000} C_DIS
LIN {X -96.447,Y -26.522,Z -51.786,A -90.000,B 90.000,C 0.000} C_DIS
LIN {X -96.499,Y -26.557,Z -51.512,A -90.000,B 90.000,C 0.000} C_DIS
LIN {X -96.537,Y -26.586,Z -51.262,A -90.000,B 90.000,C 0.000} C_DIS
LIN {X -96.552,Y -26.593,Z -51.149,A -90.000,B 90.000,C 0.000} C_DIS
LIN {X -96.568,Y -26.599,Z -51.046,A -90.000,B 90.000,C 0.000} C_DIS
LIN {X -96.578,Y -26.605,Z -50.952,A -90.000,B 90.000,C 0.000} C_DIS
LIN {X -96.583,Y -26.612,Z -50.875,A -90.000,B 90.000,C 0.000} C_DIS
LIN {X -96.591,Y -26.645,Z -50.475,A -90.000,B 90.000,C 0.000} C_DIS
LIN {X -96.588,Y -26.654,Z -50.361,A -90.000,B 90.000,C 0.000} C_DIS
LIN {X -96.575,Y -26.672,Z -50.126,A -90.000,B 90.000,C 0.000} C_DIS
LIN {X -96.560,Y -26.681,Z -49.980,A -90.000,B 90.000,C 0.000} C_DIS
LIN {X -96.533,Y -26.697,Z -49.788,A -90.000,B 90.000,C 0.000} C_DIS
LIN {X -96.523,Y -26.699,Z -49.722,A -90.000,B 90.000,C 0.000} C_DIS
LIN {X -96.514,Y -26.702,Z -49.639,A -90.000,B 90.000,C 0.000} C_DIS
LIN {X -96.494,Y -26.707,Z -49.522,A -90.000,B 90.000,C 0.000} C_DIS
LIN {X -96.457,Y -26.710,Z -49.371,A -90.000,B 90.000,C 0.000} C_DIS
LIN {X -96.388,Y -26.720,Z -49.131,A -90.000,B 90.000,C 0.000} C_DIS
LIN {X -96.351,Y -26.723,Z -49.019,A -90.000,B 90.000,C 0.000} C_DIS
LIN {X -96.310,Y -26.729,Z -48.915,A -90.000,B 90.000,C 0.000} C_DIS
LIN {X -96.195,Y -26.734,Z -48.676,A -90.000,B 90.000,C 0.000} C_DIS
LIN {X -96.163,Y -26.732,Z -48.597,A -90.000,B 90.000,C 0.000} C_DIS
LIN {X -96.123,Y -26.731,Z -48.512,A -90.000,B 90.000,C 0.000} C_DIS
LIN {X -96.029,Y -26.737,Z -48.333,A -90.000,B 90.000,C 0.000} C_DIS
LIN {X -95.938,Y -26.734,Z -48.173,A -90.000,B 90.000,C 0.000} C_DIS
LIN {X -95.886,Y -26.734,Z -48.090,A -90.000,B 90.000,C 0.000} C_DIS
LIN {X -95.813,Y -26.730,Z -47.989,A -90.000,B 90.000,C 0.000} C_DIS
LIN {X -95.652,Y -26.735,Z -47.795,A -90.000,B 90.000,C 0.000} C_DIS
LIN {X -95.593,Y -26.735,Z -47.729,A -90.000,B 90.000,C 0.000} C_DIS
LIN {X -95.544,Y -26.732,Z -47.664,A -90.000,B 90.000,C 0.000} C_DIS
LIN {X -95.467,Y -26.730,Z -47.573,A -90.000,B 90.000,C 0.000} C_DIS
LIN {X -95.396,Y -26.723,Z -47.495,A -90.000,B 90.000,C 0.000} C_DIS
LIN {X -95.290,Y -26.718,Z -47.377,A -90.000,B 90.000,C 0.000} C_DIS
LIN {X -95.187,Y -26.716,Z -47.275,A -90.000,B 90.000,C 0.000} C_DIS
LIN {X -95.088,Y -26.713,Z -47.190,A -90.000,B 90.000,C 0.000} C_DIS
LIN {X -94.970,Y -26.712,Z -47.100,A -90.000,B 90.000,C 0.000} C_DIS
LIN {X -94.854,Y -26.704,Z -47.017,A -90.000,B 90.000,C 0.000} C_DIS
LIN {X -94.768,Y -26.694,Z -46.945,A -90.000,B 90.000,C 0.000} C_DIS
LIN {X -94.644,Y -26.679,Z -46.849,A -90.000,B 90.000,C 0.000} C_DIS
LIN {X -94.567,Y -26.671,Z -46.791,A -90.000,B 90.000,C 0.000} C_DIS
LIN {X -94.371,Y -26.654,Z -46.651,A -90.000,B 90.000,C 0.000} C_DIS
LIN {X -94.284,Y -26.644,Z -46.591,A -90.000,B 90.000,C 0.000} C_DIS
LIN {X -94.135,Y -26.628,Z -46.504,A -90.000,B 90.000,C 0.000} C_DIS
LIN {X -93.997,Y -26.614,Z -46.438,A -90.000,B 90.000,C 0.000} C_DIS
LIN {X -93.783,Y -26.593,Z -46.338,A -90.000,B 90.000,C 0.000} C_DIS
LIN {X -93.606,Y -26.566,Z -46.273,A -90.000,B 90.000,C 0.000} C_DIS
LIN {X -93.446,Y -26.548,Z -46.226,A -90.000,B 90.000,C 0.000} C_DIS
LIN {X -93.215,Y -26.514,Z -46.138,A -90.000,B 90.000,C 0.000} C_DIS
LIN {X -93.090,Y -26.498,Z -46.096,A -90.000,B 90.000,C 0.000} C_DIS
LIN {X -92.972,Y -26.484,Z -46.066,A -90.000,B 90.000,C 0.000} C_DIS
LIN {X -92.662,Y -26.449,Z -45.991,A -90.000,B 90.000,C 0.000} C_DIS
LIN {X -92.523,Y -26.437,Z -45.965,A -90.000,B 90.000,C 0.000} C_DIS
LIN {X -92.279,Y -26.401,Z -45.929,A -90.000,B 90.000,C 0.000} C_DIS
LIN {X -91.975,Y -26.354,Z -45.888,A -90.000,B 90.000,C 0.000} C_DIS
LIN {X -91.859,Y -26.341,Z -45.878,A -90.000,B 90.000,C 0.000} C_DIS
LIN {X -91.516,Y -26.310,Z -45.869,A -90.000,B 90.000,C 0.000} C_DIS
LIN {X -91.444,Y -26.303,Z -45.868,A -90.000,B 90.000,C 0.000} C_DIS
LIN {X -91.267,Y -26.291,Z -45.872,A -90.000,B 90.000,C 0.000} C_DIS
LIN {X -90.899,Y -26.274,Z -45.893,A -90.000,B 90.000,C 0.000} C_DIS
LIN {X -90.539,Y -26.245,Z -45.922,A -90.000,B 90.000,C 0.000} C_DIS
LIN {X -90.399,Y -26.227,Z -45.940,A -90.000,B 90.000,C 0.000} C_DIS
LIN {X -90.066,Y -26.191,Z -45.992,A -90.000,B 90.000,C 0.000} C_DIS
LIN {X -89.758,Y -26.161,Z -46.042,A -90.000,B 90.000,C 0.000} C_DIS
LIN {X -89.534,Y -26.138,Z -46.079,A -90.000,B 90.000,C 0.000} C_DIS
LIN {X -89.197,Y -26.092,Z -46.146,A -90.000,B 90.000,C 0.000} C_DIS
LIN {X -89.092,Y -26.082,Z -46.172,A -90.000,B 90.000,C 0.000} C_DIS
LIN {X -87.976,Y -25.993,Z -46.475,A -90.000,B 90.000,C 0.000} C_DIS
LIN {X -87.853,Y -25.985,Z -46.512,A -90.000,B 90.000,C 0.000} C_DIS
LIN {X -87.541,Y -25.975,Z -46.616,A -90.000,B 90.000,C 0.000} C_DIS
LIN {X -86.935,Y -25.939,Z -46.844,A -90.000,B 90.000,C 0.000} C_DIS
LIN {X -86.322,Y -25.895,Z -47.084,A -90.000,B 90.000,C 0.000} C_DIS
LIN {X -85.931,Y -25.868,Z -47.243,A -90.000,B 90.000,C 0.000} C_DIS
LIN {X -85.153,Y -25.826,Z -47.573,A -90.000,B 90.000,C 0.000} C_DIS
LIN {X -84.931,Y -25.819,Z -47.674,A -90.000,B 90.000,C 0.000} C_DIS
LIN {X -84.835,Y -25.835,Z -47.694,A -90.000,B 90.000,C 0.000} C_DIS
LIN {X -84.562,Y -25.883,Z -47.760,A -90.000,B 90.000,C 0.000} C_DIS
LIN {X -84.268,Y -25.934,Z -47.835,A -90.000,B 90.000,C 0.000} C_DIS
LIN {X -84.167,Y -25.951,Z -47.866,A -90.000,B 90.000,C 0.000} C_DIS
LIN {X -83.272,Y -26.102,Z -48.165,A -90.000,B 90.000,C 0.000} C_DIS
LIN {X -82.974,Y -26.151,Z -48.272,A -90.000,B 90.000,C 0.000} C_DIS
LIN {X -82.351,Y -26.252,Z -48.505,A -90.000,B 90.000,C 0.000} C_DIS
LIN {X -82.058,Y -26.301,Z -48.619,A -90.000,B 90.000,C 0.000} C_DIS
LIN {X -81.959,Y -26.317,Z -48.663,A -90.000,B 90.000,C 0.000} C_DIS
LIN {X -81.152,Y -26.445,Z -49.059,A -90.000,B 90.000,C 0.000} C_DIS
LIN {X -80.888,Y -26.483,Z -49.194,A -90.000,B 90.000,C 0.000} C_DIS
LIN {X -80.274,Y -26.570,Z -49.498,A -90.000,B 90.000,C 0.000} C_DIS
LIN {X -79.896,Y -26.623,Z -49.688,A -90.000,B 90.000,C 0.000} C_DIS
LIN {X -79.806,Y -26.635,Z -49.737,A -90.000,B 90.000,C 0.000} C_DIS
LIN {X -79.766,Y -26.640,Z -49.760,A -90.000,B 90.000,C 0.000} C_DIS
LIN {X -79.531,Y -26.685,Z -49.892,A -90.000,B 90.000,C 0.000} C_DIS
LIN {X -79.025,Y -26.758,Z -50.189,A -90.000,B 90.000,C 0.000} C_DIS
LIN {X -78.910,Y -26.774,Z -50.259,A -90.000,B 90.000,C 0.000} C_DIS
LIN {X -78.384,Y -26.859,Z -50.579,A -90.000,B 90.000,C 0.000} C_DIS
LIN {X -78.220,Y -26.885,Z -50.669,A -90.000,B 90.000,C 0.000} C_DIS
LIN {X -78.118,Y -26.898,Z -50.726,A -90.000,B 90.000,C 0.000} C_DIS
LIN {X -77.891,Y -26.943,Z -50.851,A -90.000,B 90.000,C 0.000} C_DIS
LIN {X -77.848,Y -26.952,Z -50.877,A -90.000,B 90.000,C 0.000} C_DIS
LIN {X -77.745,Y -26.961,Z -50.841,A -90.000,B 90.000,C 0.000} C_DIS
LIN {X -77.731,Y -26.962,Z -50.833,A -90.000,B 90.000,C 0.000} C_DIS
LIN {X -77.494,Y -27.001,Z -50.684,A -90.000,B 90.000,C 0.000} C_DIS
LIN {X -77.348,Y -27.024,Z -50.519,A -90.000,B 90.000,C 0.000} C_DIS
LIN {X -77.280,Y -27.038,Z -50.447,A -90.000,B 90.000,C 0.000} C_DIS
LIN {X -77.376,Y -27.044,Z -49.997,A -90.000,B 90.000,C 0.000} C_DIS
LIN {X -77.398,Y -27.047,Z -49.876,A -90.000,B 90.000,C 0.000} C_DIS
LIN {X -77.418,Y -27.053,Z -49.700,A -90.000,B 90.000,C 0.000} C_DIS
LIN {X -77.447,Y -27.058,Z -49.499,A -90.000,B 90.000,C 0.000} C_DIS
LIN {X -77.454,Y -27.061,Z -49.444,A -90.000,B 90.000,C 0.000} C_DIS
LIN {X -77.631,Y -27.066,Z -49.026,A -90.000,B 90.000,C 0.000} C_DIS
LIN {X -77.686,Y -27.070,Z -48.865,A -90.000,B 90.000,C 0.000} C_DIS
LIN {X -77.701,Y -27.072,Z -48.811,A -90.000,B 90.000,C 0.000} C_DIS
LIN {X -77.729,Y -27.077,Z -48.687,A -90.000,B 90.000,C 0.000} C_DIS
LIN {X -77.737,Y -27.079,Z -48.647,A -90.000,B 90.000,C 0.000} C_DIS
LIN {X -77.758,Y -27.087,Z -48.488,A -90.000,B 90.000,C 0.000} C_DIS
LIN {X -77.766,Y -27.094,Z -48.334,A -90.000,B 90.000,C 0.000} C_DIS
LIN {X -77.758,Y -27.105,Z -48.106,A -90.000,B 90.000,C 0.000} C_DIS
LIN {X -77.754,Y -27.108,Z -48.046,A -90.000,B 90.000,C 0.000} C_DIS
LIN {X -77.709,Y -27.126,Z -47.763,A -90.000,B 90.000,C 0.000} C_DIS
LIN {X -77.677,Y -27.136,Z -47.640,A -90.000,B 90.000,C 0.000} C_DIS
LIN {X -77.660,Y -27.151,Z -47.229,A -90.000,B 90.000,C 0.000} C_DIS
LIN {X -77.647,Y -27.152,Z -47.063,A -90.000,B 90.000,C 0.000} C_DIS
LIN {X -77.635,Y -27.152,Z -46.972,A -90.000,B 90.000,C 0.000} C_DIS
LIN {X -77.625,Y -27.151,Z -46.917,A -90.000,B 90.000,C 0.000} C_DIS
LIN {X -77.596,Y -27.151,Z -46.787,A -90.000,B 90.000,C 0.000} C_DIS
LIN {X -77.567,Y -27.151,Z -46.685,A -90.000,B 90.000,C 0.000} C_DIS
LIN {X -77.543,Y -27.151,Z -46.614,A -90.000,B 90.000,C 0.000} C_DIS
LIN {X -77.472,Y -27.153,Z -46.441,A -90.000,B 90.000,C 0.000} C_DIS
LIN {X -77.352,Y -27.157,Z -46.221,A -90.000,B 90.000,C 0.000} C_DIS
LIN {X -77.282,Y -27.159,Z -46.117,A -90.000,B 90.000,C 0.000} C_DIS
LIN {X -77.202,Y -27.159,Z -46.005,A -90.000,B 90.000,C 0.000} C_DIS
LIN {X -77.106,Y -27.160,Z -45.889,A -90.000,B 90.000,C 0.000} C_DIS
LIN {X -77.052,Y -27.160,Z -45.831,A -90.000,B 90.000,C 0.000} C_DIS
LIN {X -76.947,Y -27.156,Z -45.729,A -90.000,B 90.000,C 0.000} C_DIS
LIN {X -76.872,Y -27.154,Z -45.666,A -90.000,B 90.000,C 0.000} C_DIS
LIN {X -76.759,Y -27.151,Z -45.580,A -90.000,B 90.000,C 0.000} C_DIS
